ABB RobotStudio station: MinorProjectFINAL.rspag

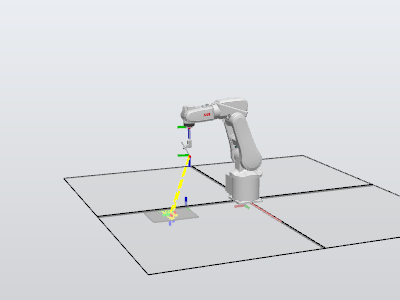
--- station ---
Station Project2 (saved by RobotStudio 23.2.10395.0)
Controller IRB120
  mechanical unit ROB_1: IRB120_3_58__01, 6 joints, base frame (0, 0, 0) mm
Layout (positions relative to the parent item):
  - IRB120_3_58__01 [mechanism, from %ABB.RobotStudio.Models.IRB120%\IRB120_3_58_G_01.rslib] at (0, 0, 0) mm; joint values [-1.5934, 0.3289, -0.2404, 0.0263, 1.472, 1.8577] (rad or m)
  - paperREVISED [part] at (105, -375, -42.57) mm, rotated rx -90 ry 0 rz 180 deg, size 210 x 3 x 297 mm
  - Part_1 [part] at (105, -375, -42.57) mm, rotated rx -90 ry 0 rz 180 deg, size 210 x 0 x 297 mm
  - Penjamin_Franklin [mechanism, from Components\Penjamin_Franklin_And his associates.rslib] at (-7.04, -394.91, 516.59) mm, rotated rx 179.86 ry -1.61 rz -17.87 deg; joint values [-0.07, 0.002] (rad or m)
Attachment: Penjamin_Franklin is attached to IRB120_3_58__01 / Link6

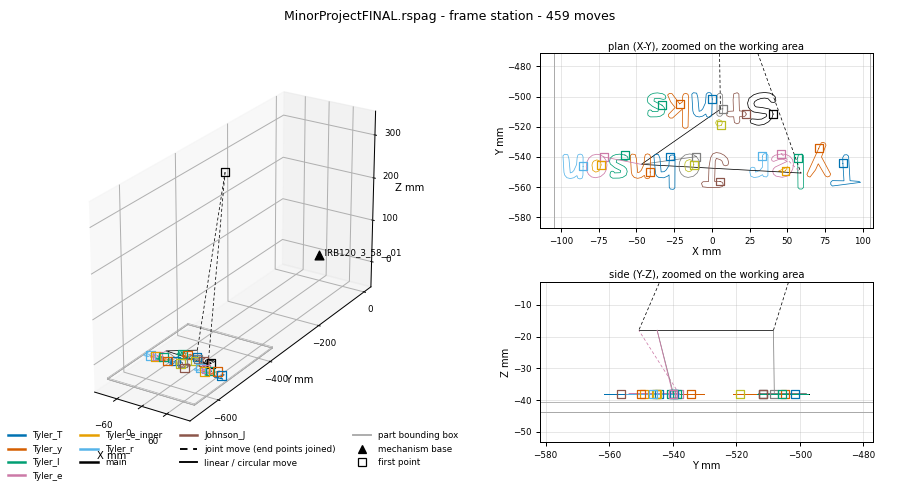
[picture p0: tool path of MinorProjectFINAL.rspag in frame station, 459 of 459 moves have a stored position in this frame; points joined in program order, loops and branches not executed]
--- Controller Data/IRB120/RAPID/TASK1/PROGMOD/CalibData.mod ---
MODULE CalibData
    PERS tooldata TCP_Pen_holder:=[TRUE,[[3.648,-1.274,111.716],[0.96514184,0.252402043,-0.069241872,0.000002181]],[0.3,[0,0,1],[1,0,0,0],0,0,0]];
    TASK PERS wobjdata Workobject_1:=[FALSE,TRUE,"",[[0,-5.508826639,-38],[0.707106781,0,0,-0.707106781]],[[375,-105,-3],[1,0,0,0]]];
    PERS tooldata My_Mechanism_1:=[TRUE,[[6.094876052,-1.40734435,179.947302726],[1,0,0,0]],[1,[1,0,0],[1,0,0,0],0,0,0]];
ENDMODULE

--- Controller Data/IRB120/RAPID/TASK1/PROGMOD/Module1.mod ---
MODULE Module1
    CONST robtarget Target_10:=[[163.751041257,191.907801073,3],[0,0.698319762,0.715785939,0],[0,0,0,0],[9E+09,9E+09,9E+09,9E+09,9E+09,9E+09]];
    CONST robtarget Target_20:=[[175.314304081,192.628796128,3],[0,0.698319762,0.715785939,0],[-1,0,1,0],[9E+09,9E+09,9E+09,9E+09,9E+09,9E+09]];
    CONST robtarget Target_30:=[[175.182166106,184.939790519,3],[0,0.698319762,0.715785939,0],[-1,0,1,0],[9E+09,9E+09,9E+09,9E+09,9E+09,9E+09]];
    CONST robtarget Target_40:=[[176.230100562,183.867034252,3],[0,0.698319762,0.715785939,0],[-1,0,1,0],[9E+09,9E+09,9E+09,9E+09,9E+09,9E+09]];
    CONST robtarget Target_50:=[[177.723746323,183.872070355,3],[0,0.698319762,0.715785939,0],[-1,0,1,0],[9E+09,9E+09,9E+09,9E+09,9E+09,9E+09]];
    CONST robtarget Target_60:=[[178.753770561,184.951832845,3],[0,0.698319762,0.715785939,0],[-1,0,1,0],[9E+09,9E+09,9E+09,9E+09,9E+09,9E+09]];
    CONST robtarget Target_70:=[[179.350705843,202.80856544,3],[0,0.698319762,0.715785939,0],[-1,0,1,0],[9E+09,9E+09,9E+09,9E+09,9E+09,9E+09]];
    CONST robtarget Target_80:=[[178.224639727,203.8775082,3],[0,0.698319762,0.715785939,0],[-1,0,1,0],[9E+09,9E+09,9E+09,9E+09,9E+09,9E+09]];
    CONST robtarget Target_90:=[[176.332276325,203.6047191,3],[0,0.698319762,0.715785939,0],[-1,0,1,0],[9E+09,9E+09,9E+09,9E+09,9E+09,9E+09]];
    CONST robtarget Target_100:=[[175.679129405,202.419661956,3],[0,0.698319762,0.715785939,0],[-1,0,1,0],[9E+09,9E+09,9E+09,9E+09,9E+09,9E+09]];
    CONST robtarget Target_110:=[[175.243917573,196.649555106,3],[0,0.698319762,0.715785939,0],[-1,0,1,0],[9E+09,9E+09,9E+09,9E+09,9E+09,9E+09]];
    CONST robtarget Target_120:=[[158.978457861,195.688923582,3],[0,0.698319762,0.715785939,0],[-1,0,1,0],[9E+09,9E+09,9E+09,9E+09,9E+09,9E+09]];
    CONST robtarget Target_130:=[[157.984185345,194.541790913,3],[0,0.698319762,0.715785939,0],[-1,0,1,0],[9E+09,9E+09,9E+09,9E+09,9E+09,9E+09]];
    CONST robtarget Target_140:=[[158.139068583,192.85150333,3],[0,0.698319762,0.715785939,0],[-1,0,1,0],[9E+09,9E+09,9E+09,9E+09,9E+09,9E+09]];
    CONST robtarget Target_150:=[[159.868914008,191.809461139,3],[0,0.698319762,0.715785939,0],[-1,0,1,0],[9E+09,9E+09,9E+09,9E+09,9E+09,9E+09]];
    CONST robtarget Target_160:=[[163.751041257,191.907801073,3],[0,0.698319762,0.715785939,0],[-1,0,1,0],[9E+09,9E+09,9E+09,9E+09,9E+09,9E+09]];
    CONST robtarget Target_170:=[[153.759568588,175.918000731,3],[0,0.698319762,0.715785939,0],[0,0,0,0],[9E+09,9E+09,9E+09,9E+09,9E+09,9E+09]];
    CONST robtarget Target_180:=[[170.978298864,168.061940799,3],[0,0.698319762,0.715785939,0],[-1,0,1,0],[9E+09,9E+09,9E+09,9E+09,9E+09,9E+09]];
    CONST robtarget Target_190:=[[172.297566022,168.691559399,3],[0,0.698319762,0.715785939,0],[-1,0,1,0],[9E+09,9E+09,9E+09,9E+09,9E+09,9E+09]];
    CONST robtarget Target_200:=[[172.832695065,170.114212978,3],[0,0.698319762,0.715785939,0],[-1,0,1,0],[9E+09,9E+09,9E+09,9E+09,9E+09,9E+09]];
    CONST robtarget Target_210:=[[168.074802834,173.749748589,3],[0,0.698319762,0.715785939,0],[-1,0,1,0],[9E+09,9E+09,9E+09,9E+09,9E+09,9E+09]];
    CONST robtarget Target_220:=[[164.005001441,175.583125337,3],[0,0.698319762,0.715785939,0],[-1,0,1,0],[9E+09,9E+09,9E+09,9E+09,9E+09,9E+09]];
    CONST robtarget Target_230:=[[172.073672363,180.31333522,3],[0,0.698319762,0.715785939,0],[-1,0,1,0],[9E+09,9E+09,9E+09,9E+09,9E+09,9E+09]];
    CONST robtarget Target_240:=[[172.764944958,181.779137598,3],[0,0.698319762,0.715785939,0],[-1,0,1,0],[9E+09,9E+09,9E+09,9E+09,9E+09,9E+09]];
    CONST robtarget Target_250:=[[172.177663158,183.183796934,3],[0,0.698319762,0.715785939,0],[-1,0,1,0],[9E+09,9E+09,9E+09,9E+09,9E+09,9E+09]];
    CONST robtarget Target_260:=[[170.825808862,183.79020191,3],[0,0.698319762,0.715785939,0],[-1,0,1,0],[9E+09,9E+09,9E+09,9E+09,9E+09,9E+09]];
    CONST robtarget Target_270:=[[159.479522834,177.713345848,3],[0,0.698319762,0.715785939,0],[-1,0,1,0],[9E+09,9E+09,9E+09,9E+09,9E+09,9E+09]];
    CONST robtarget Target_280:=[[151.640593909,180.699110514,3],[0,0.698319762,0.715785939,0],[-1,0,1,0],[9E+09,9E+09,9E+09,9E+09,9E+09,9E+09]];
    CONST robtarget Target_290:=[[150.321278848,180.083699197,3],[0,0.698319762,0.715785939,0],[-1,0,1,0],[9E+09,9E+09,9E+09,9E+09,9E+09,9E+09]];
    CONST robtarget Target_300:=[[149.800359463,178.661095912,3],[0,0.698319762,0.715785939,0],[-1,0,1,0],[9E+09,9E+09,9E+09,9E+09,9E+09,9E+09]];
    CONST robtarget Target_310:=[[150.137994684,177.553972625,3],[0,0.698319762,0.715785939,0],[-1,0,1,0],[9E+09,9E+09,9E+09,9E+09,9E+09,9E+09]];
    CONST robtarget Target_320:=[[153.759568588,175.918000731,3],[0,0.698319762,0.715785939,0],[-1,0,1,0],[9E+09,9E+09,9E+09,9E+09,9E+09,9E+09]];
    CONST robtarget Target_330:=[[160.172124107,161.930071278,3],[0,0.698319762,0.715785939,0],[0,0,0,0],[9E+09,9E+09,9E+09,9E+09,9E+09,9E+09]];
    CONST robtarget Target_340:=[[179.798680323,162.131224905,3],[0,0.698319762,0.715785939,0],[-1,0,1,0],[9E+09,9E+09,9E+09,9E+09,9E+09,9E+09]];
    CONST robtarget Target_350:=[[180.757857374,163.153918745,3],[0,0.698319762,0.715785939,0],[-1,0,1,0],[9E+09,9E+09,9E+09,9E+09,9E+09,9E+09]];
    CONST robtarget Target_360:=[[180.758005009,164.688432855,3],[0,0.698319762,0.715785939,0],[-1,0,1,0],[9E+09,9E+09,9E+09,9E+09,9E+09,9E+09]];
    CONST robtarget Target_370:=[[179.791737876,165.768569394,3],[0,0.698319762,0.715785939,0],[-1,0,1,0],[9E+09,9E+09,9E+09,9E+09,9E+09,9E+09]];
    CONST robtarget Target_380:=[[158.617763384,165.707834792,3],[0,0.698319762,0.715785939,0],[-1,0,1,0],[9E+09,9E+09,9E+09,9E+09,9E+09,9E+09]];
    CONST robtarget Target_390:=[[157.598293381,164.660075232,3],[0,0.698319762,0.715785939,0],[-1,0,1,0],[9E+09,9E+09,9E+09,9E+09,9E+09,9E+09]];
    CONST robtarget Target_400:=[[158.145784606,162.413430484,3],[0,0.698319762,0.715785939,0],[-1,0,1,0],[9E+09,9E+09,9E+09,9E+09,9E+09,9E+09]];
    CONST robtarget Target_410:=[[160.172124107,161.930071278,3],[0,0.698319762,0.715785939,0],[-1,0,1,0],[9E+09,9E+09,9E+09,9E+09,9E+09,9E+09]];
    CONST robtarget Target_420:=[[157.466190298,151.165133067,3],[0,0.698319762,0.715785939,0],[0,0,0,0],[9E+09,9E+09,9E+09,9E+09,9E+09,9E+09]];
    CONST robtarget Target_430:=[[158.332912519,146.948141754,3],[0,0.698319762,0.715785939,0],[-1,0,1,0],[9E+09,9E+09,9E+09,9E+09,9E+09,9E+09]];
    CONST robtarget Target_440:=[[159.511105335,145.172500176,3],[0,0.698319762,0.715785939,0],[-1,0,1,0],[9E+09,9E+09,9E+09,9E+09,9E+09,9E+09]];
    CONST robtarget Target_450:=[[160.983662843,144.584262074,3],[0,0.698319762,0.715785939,0],[-1,0,1,0],[9E+09,9E+09,9E+09,9E+09,9E+09,9E+09]];
    CONST robtarget Target_460:=[[162.058689867,144.95730411,3],[0,0.698319762,0.715785939,0],[-1,0,1,0],[9E+09,9E+09,9E+09,9E+09,9E+09,9E+09]];
    CONST robtarget Target_470:=[[162.413713886,146.066767593,3],[0,0.698319762,0.715785939,0],[-1,0,1,0],[9E+09,9E+09,9E+09,9E+09,9E+09,9E+09]];
    CONST robtarget Target_480:=[[161.120102459,149.419153576,3],[0,0.698319762,0.715785939,0],[-1,0,1,0],[9E+09,9E+09,9E+09,9E+09,9E+09,9E+09]];
    CONST robtarget Target_490:=[[161.007182593,152.356373467,3],[0,0.698319762,0.715785939,0],[-1,0,1,0],[9E+09,9E+09,9E+09,9E+09,9E+09,9E+09]];
    CONST robtarget Target_500:=[[162.383437332,155.046418547,3],[0,0.698319762,0.715785939,0],[-1,0,1,0],[9E+09,9E+09,9E+09,9E+09,9E+09,9E+09]];
    CONST robtarget Target_510:=[[166.147149915,147.073948161,3],[0,0.698319762,0.715785939,0],[-1,0,1,0],[9E+09,9E+09,9E+09,9E+09,9E+09,9E+09]];
    CONST robtarget Target_520:=[[167.44807257,145.7676018,3],[0,0.698319762,0.715785939,0],[-1,0,1,0],[9E+09,9E+09,9E+09,9E+09,9E+09,9E+09]];
    CONST robtarget Target_530:=[[168.923660296,145.335667719,3],[0,0.698319762,0.715785939,0],[-1,0,1,0],[9E+09,9E+09,9E+09,9E+09,9E+09,9E+09]];
    CONST robtarget Target_540:=[[170.84708047,145.878521444,3],[0,0.698319762,0.715785939,0],[-1,0,1,0],[9E+09,9E+09,9E+09,9E+09,9E+09,9E+09]];
    CONST robtarget Target_550:=[[172.184335093,147.492140687,3],[0,0.698319762,0.715785939,0],[-1,0,1,0],[9E+09,9E+09,9E+09,9E+09,9E+09,9E+09]];
    CONST robtarget Target_560:=[[172.966155304,151.601026046,3],[0,0.698319762,0.715785939,0],[-1,0,1,0],[9E+09,9E+09,9E+09,9E+09,9E+09,9E+09]];
    CONST robtarget Target_570:=[[172.266262418,154.799124826,3],[0,0.698319762,0.715785939,0],[-1,0,1,0],[9E+09,9E+09,9E+09,9E+09,9E+09,9E+09]];
    CONST robtarget Target_580:=[[170.190632557,157.260845666,3],[0,0.698319762,0.715785939,0],[-1,0,1,0],[9E+09,9E+09,9E+09,9E+09,9E+09,9E+09]];
    CONST robtarget Target_590:=[[167.422340833,158.668803926,3],[0,0.698319762,0.715785939,0],[-1,0,1,0],[9E+09,9E+09,9E+09,9E+09,9E+09,9E+09]];
    CONST robtarget Target_600:=[[164.103105526,159.130046378,3],[0,0.698319762,0.715785939,0],[-1,0,1,0],[9E+09,9E+09,9E+09,9E+09,9E+09,9E+09]];
    CONST robtarget Target_610:=[[161.217274645,158.523560707,3],[0,0.698319762,0.715785939,0],[-1,0,1,0],[9E+09,9E+09,9E+09,9E+09,9E+09,9E+09]];
    CONST robtarget Target_620:=[[159.067198932,156.726044653,3],[0,0.698319762,0.715785939,0],[-1,0,1,0],[9E+09,9E+09,9E+09,9E+09,9E+09,9E+09]];
    CONST robtarget Target_630:=[[157.860720068,154.253257576,3],[0,0.698319762,0.715785939,0],[-1,0,1,0],[9E+09,9E+09,9E+09,9E+09,9E+09,9E+09]];
    CONST robtarget Target_640:=[[157.466190298,151.165133067,3],[0,0.698319762,0.715785939,0],[-1,0,1,0],[9E+09,9E+09,9E+09,9E+09,9E+09,9E+09]];
    CONST robtarget Target_650:=[[168.639209719,153.845580268,3],[0,0.698319762,0.715785939,0],[0,0,0,0],[9E+09,9E+09,9E+09,9E+09,9E+09,9E+09]];
    CONST robtarget Target_660:=[[169.527749784,151.589432826,3],[0,0.698319762,0.715785939,0],[-1,0,1,0],[9E+09,9E+09,9E+09,9E+09,9E+09,9E+09]];
    CONST robtarget Target_670:=[[168.996213692,149.10115439,3],[0,0.698319762,0.715785939,0],[-1,0,1,0],[9E+09,9E+09,9E+09,9E+09,9E+09,9E+09]];
    CONST robtarget Target_680:=[[165.991391199,155.342751383,3],[0,0.698319762,0.715785939,0],[-1,0,1,0],[9E+09,9E+09,9E+09,9E+09,9E+09,9E+09]];
    CONST robtarget Target_690:=[[168.639209719,153.845580268,3],[0,0.698319762,0.715785939,0],[-1,0,1,0],[9E+09,9E+09,9E+09,9E+09,9E+09,9E+09]];
    CONST robtarget Target_700:=[[159.08585114,138.553482656,3],[0,0.698319762,0.715785939,0],[0,0,0,0],[9E+09,9E+09,9E+09,9E+09,9E+09,9E+09]];
    CONST robtarget Target_710:=[[166.232578876,138.591784231,3],[0,0.698319762,0.715785939,0],[-1,0,1,0],[9E+09,9E+09,9E+09,9E+09,9E+09,9E+09]];
    CONST robtarget Target_720:=[[168.444594894,136.76635106,3],[0,0.698319762,0.715785939,0],[-1,0,1,0],[9E+09,9E+09,9E+09,9E+09,9E+09,9E+09]];
    CONST robtarget Target_730:=[[169.530122845,134.02777656,3],[0,0.698319762,0.715785939,0],[-1,0,1,0],[9E+09,9E+09,9E+09,9E+09,9E+09,9E+09]];
    CONST robtarget Target_740:=[[166.711519604,133.499671613,3],[0,0.698319762,0.715785939,0],[-1,0,1,0],[9E+09,9E+09,9E+09,9E+09,9E+09,9E+09]];
    CONST robtarget Target_750:=[[166.254280251,132.15542517,3],[0,0.698319762,0.715785939,0],[-1,0,1,0],[9E+09,9E+09,9E+09,9E+09,9E+09,9E+09]];
    CONST robtarget Target_760:=[[166.802526185,130.739972078,3],[0,0.698319762,0.715785939,0],[-1,0,1,0],[9E+09,9E+09,9E+09,9E+09,9E+09,9E+09]];
    CONST robtarget Target_770:=[[169.386818084,130.176801905,3],[0,0.698319762,0.715785939,0],[-1,0,1,0],[9E+09,9E+09,9E+09,9E+09,9E+09,9E+09]];
    CONST robtarget Target_780:=[[172.218984231,130.896775724,3],[0,0.698319762,0.715785939,0],[-1,0,1,0],[9E+09,9E+09,9E+09,9E+09,9E+09,9E+09]];
    CONST robtarget Target_790:=[[173.156645819,133.031201627,3],[0,0.698319762,0.715785939,0],[-1,0,1,0],[9E+09,9E+09,9E+09,9E+09,9E+09,9E+09]];
    CONST robtarget Target_800:=[[172.677884374,135.960083101,3],[0,0.698319762,0.715785939,0],[-1,0,1,0],[9E+09,9E+09,9E+09,9E+09,9E+09,9E+09]];
    CONST robtarget Target_810:=[[171.262323998,138.608742947,3],[0,0.698319762,0.715785939,0],[-1,0,1,0],[9E+09,9E+09,9E+09,9E+09,9E+09,9E+09]];
    CONST robtarget Target_820:=[[172.475042596,139.230902153,3],[0,0.698319762,0.715785939,0],[-1,0,1,0],[9E+09,9E+09,9E+09,9E+09,9E+09,9E+09]];
    CONST robtarget Target_830:=[[172.739912492,141.268936192,3],[0,0.698319762,0.715785939,0],[-1,0,1,0],[9E+09,9E+09,9E+09,9E+09,9E+09,9E+09]];
    CONST robtarget Target_840:=[[171.738633757,142.199761024,3],[0,0.698319762,0.715785939,0],[-1,0,1,0],[9E+09,9E+09,9E+09,9E+09,9E+09,9E+09]];
    CONST robtarget Target_850:=[[158.348865178,142.216780556,3],[0,0.698319762,0.715785939,0],[-1,0,1,0],[9E+09,9E+09,9E+09,9E+09,9E+09,9E+09]];
    CONST robtarget Target_860:=[[157.343188099,141.289841504,3],[0,0.698319762,0.715785939,0],[-1,0,1,0],[9E+09,9E+09,9E+09,9E+09,9E+09,9E+09]];
    CONST robtarget Target_870:=[[157.339567123,139.730448483,3],[0,0.698319762,0.715785939,0],[-1,0,1,0],[9E+09,9E+09,9E+09,9E+09,9E+09,9E+09]];
    CONST robtarget Target_880:=[[158.344774317,138.689520265,3],[0,0.698319762,0.715785939,0],[-1,0,1,0],[9E+09,9E+09,9E+09,9E+09,9E+09,9E+09]];
    CONST robtarget Target_890:=[[159.08585114,138.553482656,3],[0,0.698319762,0.715785939,0],[-1,0,1,0],[9E+09,9E+09,9E+09,9E+09,9E+09,9E+09]];
    CONST robtarget Homes:=[[3.863516215,-397.404717523,336.886300892],[0.003386746,0.987758585,-0.155352434,0.013679542],[-2,0,1,0],[9E+09,9E+09,9E+09,9E+09,9E+09,9E+09]];
    CONST robtarget liftPoint_Tyler:=[[170.167,164.128,23],[0,0.698319762,0.715785939,0],[-1,0,1,0],[9E+09,9E+09,9E+09,9E+09,9E+09,9E+09]];
    CONST robtarget Target_900:=[[175.775906994,110.505400925,3],[0,0.698319762,0.715785939,0],[-2,1,-1,0],[9E+09,9E+09,9E+09,9E+09,9E+09,9E+09]];
    CONST robtarget Target_910:=[[175.731485499,106.825258538,3],[0,0.698319762,0.715785939,0],[-2,1,-1,0],[9E+09,9E+09,9E+09,9E+09,9E+09,9E+09]];
    CONST robtarget Target_920:=[[162.3172094,107.263116295,3],[0,0.698319762,0.715785939,0],[-2,1,-1,0],[9E+09,9E+09,9E+09,9E+09,9E+09,9E+09]];
    CONST robtarget Target_930:=[[160.425013825,107.99558071,3],[0,0.698319762,0.715785939,0],[-2,1,-1,0],[9E+09,9E+09,9E+09,9E+09,9E+09,9E+09]];
    CONST robtarget Target_940:=[[161.374954401,110.705498367,3],[0,0.698319762,0.715785939,0],[-2,1,-1,0],[9E+09,9E+09,9E+09,9E+09,9E+09,9E+09]];
    CONST robtarget Target_950:=[[162.300171542,111.790233782,3],[0,0.698319762,0.715785939,0],[-2,1,-1,0],[9E+09,9E+09,9E+09,9E+09,9E+09,9E+09]];
    CONST robtarget Target_960:=[[164.806818321,112.660077554,3],[0,0.698319762,0.715785939,0],[-2,1,-1,0],[9E+09,9E+09,9E+09,9E+09,9E+09,9E+09]];
    CONST robtarget Target_970:=[[165.348767223,114.164446335,3],[0,0.698319762,0.715785939,0],[-2,1,-1,0],[9E+09,9E+09,9E+09,9E+09,9E+09,9E+09]];
    CONST robtarget Target_980:=[[164.789571873,115.665102404,3],[0,0.698319762,0.715785939,0],[-2,1,-1,0],[9E+09,9E+09,9E+09,9E+09,9E+09,9E+09]];
    CONST robtarget Target_990:=[[163.125514309,116.16034525,3],[0,0.698319762,0.715785939,0],[-2,1,-1,0],[9E+09,9E+09,9E+09,9E+09,9E+09,9E+09]];
    CONST robtarget Target_1000:=[[160.563384619,115.419967167,3],[0,0.698319762,0.715785939,0],[-2,1,-1,0],[9E+09,9E+09,9E+09,9E+09,9E+09,9E+09]];
    CONST robtarget Target_1010:=[[158.361392746,113.217334114,3],[0,0.698319762,0.715785939,0],[-2,1,-1,0],[9E+09,9E+09,9E+09,9E+09,9E+09,9E+09]];
    CONST robtarget Target_1020:=[[157.00616506,110.612614131,3],[0,0.698319762,0.715785939,0],[-2,1,-1,0],[9E+09,9E+09,9E+09,9E+09,9E+09,9E+09]];
    CONST robtarget Target_1030:=[[156.560356456,107.982550303,3],[0,0.698319762,0.715785939,0],[-2,1,-1,0],[9E+09,9E+09,9E+09,9E+09,9E+09,9E+09]];
    CONST robtarget Target_1040:=[[157.424300306,105.644618187,3],[0,0.698319762,0.715785939,0],[-2,1,-1,0],[9E+09,9E+09,9E+09,9E+09,9E+09,9E+09]];
    CONST robtarget Target_1050:=[[159.997448553,104.172057738,3],[0,0.698319762,0.715785939,0],[-2,1,-1,0],[9E+09,9E+09,9E+09,9E+09,9E+09,9E+09]];
    CONST robtarget Target_1060:=[[166.0289515,103.116099725,3],[0,0.698319762,0.715785939,0],[-2,1,-1,0],[9E+09,9E+09,9E+09,9E+09,9E+09,9E+09]];
    CONST robtarget Target_1070:=[[175.830387142,102.776182007,3],[0,0.698319762,0.715785939,0],[-2,1,-1,0],[9E+09,9E+09,9E+09,9E+09,9E+09,9E+09]];
    CONST robtarget Target_1080:=[[175.902977488,99.156821148,3],[0,0.698319762,0.715785939,0],[-2,1,-1,0],[9E+09,9E+09,9E+09,9E+09,9E+09,9E+09]];
    CONST robtarget Target_1090:=[[177.007630849,98.11977592,3],[0,0.698319762,0.715785939,0],[-2,1,-1,0],[9E+09,9E+09,9E+09,9E+09,9E+09,9E+09]];
    CONST robtarget Target_1100:=[[179.292389298,98.951563604,3],[0,0.698319762,0.715785939,0],[-2,1,-1,0],[9E+09,9E+09,9E+09,9E+09,9E+09,9E+09]];
    CONST robtarget Target_1110:=[[179.783379524,102.926267927,3],[0,0.698319762,0.715785939,0],[-2,1,-1,0],[9E+09,9E+09,9E+09,9E+09,9E+09,9E+09]];
    CONST robtarget Target_1120:=[[179.656450737,110.021188597,3],[0,0.698319762,0.715785939,0],[-2,1,-1,0],[9E+09,9E+09,9E+09,9E+09,9E+09,9E+09]];
    CONST robtarget Target_1130:=[[179.166938366,111.927031105,3],[0,0.698319762,0.715785939,0],[-2,1,-1,0],[9E+09,9E+09,9E+09,9E+09,9E+09,9E+09]];
    CONST robtarget Target_1140:=[[177.715551642,112.557965304,3],[0,0.698319762,0.715785939,0],[-2,1,-1,0],[9E+09,9E+09,9E+09,9E+09,9E+09,9E+09]];
    CONST robtarget Target_1150:=[[176.282616704,111.927958684,3],[0,0.698319762,0.715785939,0],[-2,1,-1,0],[9E+09,9E+09,9E+09,9E+09,9E+09,9E+09]];
    CONST robtarget Target_1160:=[[175.775906994,110.505400925,3],[0,0.698319762,0.715785939,0],[-2,1,-1,0],[9E+09,9E+09,9E+09,9E+09,9E+09,9E+09]];
    CONST robtarget Target_1170:=[[159.276068814,94.777825568,3],[0,0.698319762,0.715785939,0],[-2,1,-1,0],[9E+09,9E+09,9E+09,9E+09,9E+09,9E+09]];
    CONST robtarget Target_1180:=[[157.929711577,92.698841911,3],[0,0.698319762,0.715785939,0],[-2,1,-1,0],[9E+09,9E+09,9E+09,9E+09,9E+09,9E+09]];
    CONST robtarget Target_1190:=[[157.486846922,90.253496701,3],[0,0.698319762,0.715785939,0],[-2,1,-1,0],[9E+09,9E+09,9E+09,9E+09,9E+09,9E+09]];
    CONST robtarget Target_1200:=[[158.146958921,87.268396908,3],[0,0.698319762,0.715785939,0],[-2,1,-1,0],[9E+09,9E+09,9E+09,9E+09,9E+09,9E+09]];
    CONST robtarget Target_1210:=[[160.104836866,84.962563313,3],[0,0.698319762,0.715785939,0],[-2,1,-1,0],[9E+09,9E+09,9E+09,9E+09,9E+09,9E+09]];
    CONST robtarget Target_1220:=[[162.680993817,83.649859269,3],[0,0.698319762,0.715785939,0],[-2,1,-1,0],[9E+09,9E+09,9E+09,9E+09,9E+09,9E+09]];
    CONST robtarget Target_1230:=[[165.737271089,83.219707087,3],[0,0.698319762,0.715785939,0],[-2,1,-1,0],[9E+09,9E+09,9E+09,9E+09,9E+09,9E+09]];
    CONST robtarget Target_1240:=[[168.517281523,83.60561224,3],[0,0.698319762,0.715785939,0],[-2,1,-1,0],[9E+09,9E+09,9E+09,9E+09,9E+09,9E+09]];
    CONST robtarget Target_1250:=[[170.804557641,84.742891106,3],[0,0.698319762,0.715785939,0],[-2,1,-1,0],[9E+09,9E+09,9E+09,9E+09,9E+09,9E+09]];
    CONST robtarget Target_1260:=[[172.502920539,86.716487904,3],[0,0.698319762,0.715785939,0],[-2,1,-1,0],[9E+09,9E+09,9E+09,9E+09,9E+09,9E+09]];
    CONST robtarget Target_1270:=[[173.062650846,89.26880086,3],[0,0.698319762,0.715785939,0],[-2,1,-1,0],[9E+09,9E+09,9E+09,9E+09,9E+09,9E+09]];
    CONST robtarget Target_1280:=[[172.326476842,92.694110719,3],[0,0.698319762,0.715785939,0],[-2,1,-1,0],[9E+09,9E+09,9E+09,9E+09,9E+09,9E+09]];
    CONST robtarget Target_1290:=[[170.143891247,95.269135257,3],[0,0.698319762,0.715785939,0],[-2,1,-1,0],[9E+09,9E+09,9E+09,9E+09,9E+09,9E+09]];
    CONST robtarget Target_1300:=[[167.510845294,96.599405006,3],[0,0.698319762,0.715785939,0],[-2,1,-1,0],[9E+09,9E+09,9E+09,9E+09,9E+09,9E+09]];
    CONST robtarget Target_1310:=[[164.540029593,96.969467873,3],[0,0.698319762,0.715785939,0],[-2,1,-1,0],[9E+09,9E+09,9E+09,9E+09,9E+09,9E+09]];
    CONST robtarget Target_1320:=[[161.576033584,96.366266342,3],[0,0.698319762,0.715785939,0],[-2,1,-1,0],[9E+09,9E+09,9E+09,9E+09,9E+09,9E+09]];
    CONST robtarget Target_1330:=[[159.276068814,94.777825568,3],[0,0.698319762,0.715785939,0],[-2,1,-1,0],[9E+09,9E+09,9E+09,9E+09,9E+09,9E+09]];
    CONST robtarget Target_1340:=[[164.553299553,93.033762171,3],[0,0.698319762,0.715785939,0],[-2,1,-1,0],[9E+09,9E+09,9E+09,9E+09,9E+09,9E+09]];
    CONST robtarget Target_1350:=[[167.710414693,92.191903115,3],[0,0.698319762,0.715785939,0],[-2,1,-1,0],[9E+09,9E+09,9E+09,9E+09,9E+09,9E+09]];
    CONST robtarget Target_1360:=[[168.915041174,91.002453619,3],[0,0.698319762,0.715785939,0],[-2,1,-1,0],[9E+09,9E+09,9E+09,9E+09,9E+09,9E+09]];
    CONST robtarget Target_1370:=[[169.3110385,89.440860296,3],[0,0.698319762,0.715785939,0],[-2,1,-1,0],[9E+09,9E+09,9E+09,9E+09,9E+09,9E+09]];
    CONST robtarget Target_1380:=[[168.162996215,87.543715835,3],[0,0.698319762,0.715785939,0],[-2,1,-1,0],[9E+09,9E+09,9E+09,9E+09,9E+09,9E+09]];
    CONST robtarget Target_1390:=[[164.729851,87.024181912,3],[0,0.698319762,0.715785939,0],[-2,1,-1,0],[9E+09,9E+09,9E+09,9E+09,9E+09,9E+09]];
    CONST robtarget Target_1400:=[[163.226272679,87.33169039,3],[0,0.698319762,0.715785939,0],[-2,1,-1,0],[9E+09,9E+09,9E+09,9E+09,9E+09,9E+09]];
    CONST robtarget Target_1410:=[[162.06916418,88.1234726,3],[0,0.698319762,0.715785939,0],[-2,1,-1,0],[9E+09,9E+09,9E+09,9E+09,9E+09,9E+09]];
    CONST robtarget Target_1420:=[[161.223636366,90.266095978,3],[0,0.698319762,0.715785939,0],[-2,1,-1,0],[9E+09,9E+09,9E+09,9E+09,9E+09,9E+09]];
    CONST robtarget Target_1430:=[[161.942226456,92.058785513,3],[0,0.698319762,0.715785939,0],[-2,1,-1,0],[9E+09,9E+09,9E+09,9E+09,9E+09,9E+09]];
    CONST robtarget Target_1440:=[[163.0480419,92.787138913,3],[0,0.698319762,0.715785939,0],[-2,1,-1,0],[9E+09,9E+09,9E+09,9E+09,9E+09,9E+09]];
    CONST robtarget Target_1450:=[[164.553299553,93.033762171,3],[0,0.698319762,0.715785939,0],[-2,1,-1,0],[9E+09,9E+09,9E+09,9E+09,9E+09,9E+09]];
    CONST robtarget Target_1460:=[[159.19401738,76.974331877,3],[0,0.698319762,0.715785939,0],[-2,1,-1,0],[9E+09,9E+09,9E+09,9E+09,9E+09,9E+09]];
    CONST robtarget Target_1470:=[[165.390517427,76.497928224,3],[0,0.698319762,0.715785939,0],[-2,1,-1,0],[9E+09,9E+09,9E+09,9E+09,9E+09,9E+09]];
    CONST robtarget Target_1480:=[[168.152961856,74.716975641,3],[0,0.698319762,0.715785939,0],[-2,1,-1,0],[9E+09,9E+09,9E+09,9E+09,9E+09,9E+09]];
    CONST robtarget Target_1490:=[[169.244459454,73.367307985,3],[0,0.698319762,0.715785939,0],[-2,1,-1,0],[9E+09,9E+09,9E+09,9E+09,9E+09,9E+09]];
    CONST robtarget Target_1500:=[[169.418127554,71.375151118,3],[0,0.698319762,0.715785939,0],[-2,1,-1,0],[9E+09,9E+09,9E+09,9E+09,9E+09,9E+09]];
    CONST robtarget Target_1510:=[[160.31671931,70.584304991,3],[0,0.698319762,0.715785939,0],[-2,1,-1,0],[9E+09,9E+09,9E+09,9E+09,9E+09,9E+09]];
    CONST robtarget Target_1520:=[[157.86917958,69.570807458,3],[0,0.698319762,0.715785939,0],[-2,1,-1,0],[9E+09,9E+09,9E+09,9E+09,9E+09,9E+09]];
    CONST robtarget Target_1530:=[[157.650162968,67.628834824,3],[0,0.698319762,0.715785939,0],[-2,1,-1,0],[9E+09,9E+09,9E+09,9E+09,9E+09,9E+09]];
    CONST robtarget Target_1540:=[[158.630714107,66.523869711,3],[0,0.698319762,0.715785939,0],[-2,1,-1,0],[9E+09,9E+09,9E+09,9E+09,9E+09,9E+09]];
    CONST robtarget Target_1550:=[[170.77309542,67.735242064,3],[0,0.698319762,0.715785939,0],[-2,1,-1,0],[9E+09,9E+09,9E+09,9E+09,9E+09,9E+09]];
    CONST robtarget Target_1560:=[[172.067452503,68.378991271,3],[0,0.698319762,0.715785939,0],[-2,1,-1,0],[9E+09,9E+09,9E+09,9E+09,9E+09,9E+09]];
    CONST robtarget Target_1570:=[[173.085710436,69.789063982,3],[0,0.698319762,0.715785939,0],[-2,1,-1,0],[9E+09,9E+09,9E+09,9E+09,9E+09,9E+09]];
    CONST robtarget Target_1580:=[[173.289145178,73.187338868,3],[0,0.698319762,0.715785939,0],[-2,1,-1,0],[9E+09,9E+09,9E+09,9E+09,9E+09,9E+09]];
    CONST robtarget Target_1590:=[[172.26880383,75.560268231,3],[0,0.698319762,0.715785939,0],[-2,1,-1,0],[9E+09,9E+09,9E+09,9E+09,9E+09,9E+09]];
    CONST robtarget Target_1600:=[[171.371831589,76.63176442,3],[0,0.698319762,0.715785939,0],[-2,1,-1,0],[9E+09,9E+09,9E+09,9E+09,9E+09,9E+09]];
    CONST robtarget Target_1610:=[[179.626520965,76.759055892,3],[0,0.698319762,0.715785939,0],[-2,0,-1,0],[9E+09,9E+09,9E+09,9E+09,9E+09,9E+09]];
    CONST robtarget Target_1620:=[[180.753677289,77.476828643,3],[0,0.698319762,0.715785939,0],[-2,0,-1,0],[9E+09,9E+09,9E+09,9E+09,9E+09,9E+09]];
    CONST robtarget Target_1630:=[[180.994004844,79.417099286,3],[0,0.698319762,0.715785939,0],[-2,0,-1,0],[9E+09,9E+09,9E+09,9E+09,9E+09,9E+09]];
    CONST robtarget Target_1640:=[[180.009982837,80.493623504,3],[0,0.698319762,0.715785939,0],[-2,0,-1,0],[9E+09,9E+09,9E+09,9E+09,9E+09,9E+09]];
    CONST robtarget Target_1650:=[[159.144449473,80.613311259,3],[0,0.698319762,0.715785939,0],[-2,1,-1,0],[9E+09,9E+09,9E+09,9E+09,9E+09,9E+09]];
    CONST robtarget Target_1660:=[[158.153655217,79.483941873,3],[0,0.698319762,0.715785939,0],[-2,1,-1,0],[9E+09,9E+09,9E+09,9E+09,9E+09,9E+09]];
    CONST robtarget Target_1670:=[[158.317789462,77.688907073,3],[0,0.698319762,0.715785939,0],[-2,1,-1,0],[9E+09,9E+09,9E+09,9E+09,9E+09,9E+09]];
    CONST robtarget Target_1680:=[[159.19401738,76.974331877,3],[0,0.698319762,0.715785939,0],[-2,1,-1,0],[9E+09,9E+09,9E+09,9E+09,9E+09,9E+09]];
    CONST robtarget Target_1690:=[[169.48675747,64.121961466,3],[0,0.698319762,0.715785939,0],[-2,1,-1,0],[9E+09,9E+09,9E+09,9E+09,9E+09,9E+09]];
    CONST robtarget Target_1700:=[[159.313738911,64.314999427,3],[0,0.698319762,0.715785939,0],[-2,0,0,0],[9E+09,9E+09,9E+09,9E+09,9E+09,9E+09]];
    CONST robtarget Target_1710:=[[157.948274945,63.756259901,3],[0,0.698319762,0.715785939,0],[-2,0,0,0],[9E+09,9E+09,9E+09,9E+09,9E+09,9E+09]];
    CONST robtarget Target_1720:=[[157.410437254,62.347807017,3],[0,0.698319762,0.715785939,0],[-2,0,0,0],[9E+09,9E+09,9E+09,9E+09,9E+09,9E+09]];
    CONST robtarget Target_1730:=[[157.961112555,60.935928878,3],[0,0.698319762,0.715785939,0],[-2,0,0,0],[9E+09,9E+09,9E+09,9E+09,9E+09,9E+09]];
    CONST robtarget Target_1740:=[[159.849926153,60.357968251,3],[0,0.698319762,0.715785939,0],[-2,0,0,0],[9E+09,9E+09,9E+09,9E+09,9E+09,9E+09]];
    CONST robtarget Target_1750:=[[164.36181293,60.013090517,3],[0,0.698319762,0.715785939,0],[-2,0,0,0],[9E+09,9E+09,9E+09,9E+09,9E+09,9E+09]];
    CONST robtarget Target_1760:=[[168.334661535,58.194362031,3],[0,0.698319762,0.715785939,0],[-2,0,0,0],[9E+09,9E+09,9E+09,9E+09,9E+09,9E+09]];
    CONST robtarget Target_1770:=[[169.512242363,57.016017545,3],[0,0.698319762,0.715785939,0],[-2,0,0,0],[9E+09,9E+09,9E+09,9E+09,9E+09,9E+09]];
    CONST robtarget Target_1780:=[[169.907511332,55.81187047,3],[0,0.698319762,0.715785939,0],[-2,0,0,0],[9E+09,9E+09,9E+09,9E+09,9E+09,9E+09]];
    CONST robtarget Target_1790:=[[160.621604004,54.956028888,3],[0,0.698319762,0.715785939,0],[-2,0,0,0],[9E+09,9E+09,9E+09,9E+09,9E+09,9E+09]];
    CONST robtarget Target_1800:=[[157.867842537,54.161722596,3],[0,0.698319762,0.715785939,0],[-2,0,0,0],[9E+09,9E+09,9E+09,9E+09,9E+09,9E+09]];
    CONST robtarget Target_1810:=[[157.57665402,52.029476397,3],[0,0.698319762,0.715785939,0],[-2,0,0,0],[9E+09,9E+09,9E+09,9E+09,9E+09,9E+09]];
    CONST robtarget Target_1820:=[[158.56772102,50.970723913,3],[0,0.698319762,0.715785939,0],[-2,0,0,0],[9E+09,9E+09,9E+09,9E+09,9E+09,9E+09]];
    CONST robtarget Target_1830:=[[169.548626817,51.632923283,3],[0,0.698319762,0.715785939,0],[-2,0,0,0],[9E+09,9E+09,9E+09,9E+09,9E+09,9E+09]];
    CONST robtarget Target_1840:=[[171.425954171,52.150759167,3],[0,0.698319762,0.715785939,0],[-2,0,0,0],[9E+09,9E+09,9E+09,9E+09,9E+09,9E+09]];
    CONST robtarget Target_1850:=[[173.104796596,53.595026505,3],[0,0.698319762,0.715785939,0],[-2,0,0,0],[9E+09,9E+09,9E+09,9E+09,9E+09,9E+09]];
    CONST robtarget Target_1860:=[[173.658368222,55.866698432,3],[0,0.698319762,0.715785939,0],[-2,0,0,0],[9E+09,9E+09,9E+09,9E+09,9E+09,9E+09]];
    CONST robtarget Target_1870:=[[173.128646274,58.109855405,3],[0,0.698319762,0.715785939,0],[-2,0,0,0],[9E+09,9E+09,9E+09,9E+09,9E+09,9E+09]];
    CONST robtarget Target_1880:=[[171.711231833,60.250550561,3],[0,0.698319762,0.715785939,0],[-2,0,0,0],[9E+09,9E+09,9E+09,9E+09,9E+09,9E+09]];
    CONST robtarget Target_1890:=[[173.382360872,60.817425607,3],[0,0.698319762,0.715785939,0],[-2,0,0,0],[9E+09,9E+09,9E+09,9E+09,9E+09,9E+09]];
    CONST robtarget Target_1900:=[[173.935223307,62.247234355,3],[0,0.698319762,0.715785939,0],[-2,0,0,0],[9E+09,9E+09,9E+09,9E+09,9E+09,9E+09]];
    CONST robtarget Target_1910:=[[173.402314827,63.659181935,3],[0,0.698319762,0.715785939,0],[-2,0,0,0],[9E+09,9E+09,9E+09,9E+09,9E+09,9E+09]];
    CONST robtarget Target_1920:=[[171.53202662,64.215880745,3],[0,0.698319762,0.715785939,0],[-2,0,0,0],[9E+09,9E+09,9E+09,9E+09,9E+09,9E+09]];
    CONST robtarget Target_1930:=[[169.48675747,64.121961466,3],[0,0.698319762,0.715785939,0],[-2,0,0,0],[9E+09,9E+09,9E+09,9E+09,9E+09,9E+09]];
    CONST robtarget Target_1940:=[[158.199861844,47.346320771,3],[0,0.698319762,0.715785939,0],[-2,1,-1,0],[9E+09,9E+09,9E+09,9E+09,9E+09,9E+09]];
    CONST robtarget Target_1950:=[[157.628963899,43.891731909,3],[0,0.698319762,0.715785939,0],[-2,1,-1,0],[9E+09,9E+09,9E+09,9E+09,9E+09,9E+09]];
    CONST robtarget Target_1960:=[[157.889451747,41.431010202,3],[0,0.698319762,0.715785939,0],[-2,1,-1,0],[9E+09,9E+09,9E+09,9E+09,9E+09,9E+09]];
    CONST robtarget Target_1970:=[[158.652931475,39.391107595,3],[0,0.698319762,0.715785939,0],[-2,1,-1,0],[9E+09,9E+09,9E+09,9E+09,9E+09,9E+09]];
    CONST robtarget Target_1980:=[[160.218043244,37.691376952,3],[0,0.698319762,0.715785939,0],[-2,1,-1,0],[9E+09,9E+09,9E+09,9E+09,9E+09,9E+09]];
    CONST robtarget Target_1990:=[[162.368966498,37.130293285,3],[0,0.698319762,0.715785939,0],[-2,1,-1,0],[9E+09,9E+09,9E+09,9E+09,9E+09,9E+09]];
    CONST robtarget Target_2000:=[[164.146814192,37.65135098,3],[0,0.698319762,0.715785939,0],[-2,0,-1,0],[9E+09,9E+09,9E+09,9E+09,9E+09,9E+09]];
    CONST robtarget Target_2010:=[[166.591204245,40.654032626,3],[0,0.698319762,0.715785939,0],[-2,0,-1,0],[9E+09,9E+09,9E+09,9E+09,9E+09,9E+09]];
    CONST robtarget Target_2020:=[[168.570761932,44.56446156,3],[0,0.698319762,0.715785939,0],[-2,0,-1,0],[9E+09,9E+09,9E+09,9E+09,9E+09,9E+09]];
    CONST robtarget Target_2030:=[[169.925253649,44.228030753,3],[0,0.698319762,0.715785939,0],[-2,0,-1,0],[9E+09,9E+09,9E+09,9E+09,9E+09,9E+09]];
    CONST robtarget Target_2040:=[[170.072823228,40.495253612,3],[0,0.698319762,0.715785939,0],[-2,0,-1,0],[9E+09,9E+09,9E+09,9E+09,9E+09,9E+09]];
    CONST robtarget Target_2050:=[[169.190256749,39.927508735,3],[0,0.698319762,0.715785939,0],[-2,0,-1,0],[9E+09,9E+09,9E+09,9E+09,9E+09,9E+09]];
    CONST robtarget Target_2060:=[[168.899236118,38.800498766,3],[0,0.698319762,0.715785939,0],[-2,0,-1,0],[9E+09,9E+09,9E+09,9E+09,9E+09,9E+09]];
    CONST robtarget Target_2070:=[[169.54208954,37.768991872,3],[0,0.698319762,0.715785939,0],[-2,0,-1,0],[9E+09,9E+09,9E+09,9E+09,9E+09,9E+09]];
    CONST robtarget Target_2080:=[[171.461375012,37.430917682,3],[0,0.698319762,0.715785939,0],[-2,0,-1,0],[9E+09,9E+09,9E+09,9E+09,9E+09,9E+09]];
    CONST robtarget Target_2090:=[[172.586600524,37.669145141,3],[0,0.698319762,0.715785939,0],[-2,0,-1,0],[9E+09,9E+09,9E+09,9E+09,9E+09,9E+09]];
    CONST robtarget Target_2100:=[[173.565226295,39.242449563,3],[0,0.698319762,0.715785939,0],[-2,0,-1,0],[9E+09,9E+09,9E+09,9E+09,9E+09,9E+09]];
    CONST robtarget Target_2110:=[[173.497108354,43.639751601,3],[0,0.698319762,0.715785939,0],[-2,0,-1,0],[9E+09,9E+09,9E+09,9E+09,9E+09,9E+09]];
    CONST robtarget Target_2120:=[[173.052668328,45.87610074,3],[0,0.698319762,0.715785939,0],[-2,0,-1,0],[9E+09,9E+09,9E+09,9E+09,9E+09,9E+09]];
    CONST robtarget Target_2130:=[[171.585119959,48.14094855,3],[0,0.698319762,0.715785939,0],[-2,0,-1,0],[9E+09,9E+09,9E+09,9E+09,9E+09,9E+09]];
    CONST robtarget Target_2140:=[[169.192007177,48.889472011,3],[0,0.698319762,0.715785939,0],[-2,0,-1,0],[9E+09,9E+09,9E+09,9E+09,9E+09,9E+09]];
    CONST robtarget Target_2150:=[[167.328853508,48.382355593,3],[0,0.698319762,0.715785939,0],[-2,0,-1,0],[9E+09,9E+09,9E+09,9E+09,9E+09,9E+09]];
    CONST robtarget Target_2160:=[[165.774565999,46.874573525,3],[0,0.698319762,0.715785939,0],[-2,1,-1,0],[9E+09,9E+09,9E+09,9E+09,9E+09,9E+09]];
    CONST robtarget Target_2170:=[[163.08914292,41.611926335,3],[0,0.698319762,0.715785939,0],[-2,1,-1,0],[9E+09,9E+09,9E+09,9E+09,9E+09,9E+09]];
    CONST robtarget Target_2180:=[[161.450867277,41.83728845,3],[0,0.698319762,0.715785939,0],[-2,1,-1,0],[9E+09,9E+09,9E+09,9E+09,9E+09,9E+09]];
    CONST robtarget Target_2190:=[[161.252557642,44.813302229,3],[0,0.698319762,0.715785939,0],[-2,1,-1,0],[9E+09,9E+09,9E+09,9E+09,9E+09,9E+09]];
    CONST robtarget Target_2200:=[[161.963575987,47.799477353,3],[0,0.698319762,0.715785939,0],[-2,1,-1,0],[9E+09,9E+09,9E+09,9E+09,9E+09,9E+09]];
    CONST robtarget Target_2210:=[[161.604087321,49.066373217,3],[0,0.698319762,0.715785939,0],[-2,1,-1,0],[9E+09,9E+09,9E+09,9E+09,9E+09,9E+09]];
    CONST robtarget Target_2220:=[[160.537042008,49.485484483,3],[0,0.698319762,0.715785939,0],[-2,1,-1,0],[9E+09,9E+09,9E+09,9E+09,9E+09,9E+09]];
    CONST robtarget Target_2230:=[[159.178401202,48.948082705,3],[0,0.698319762,0.715785939,0],[-2,1,-1,0],[9E+09,9E+09,9E+09,9E+09,9E+09,9E+09]];
    CONST robtarget Target_2240:=[[158.199861844,47.346320771,3],[0,0.698319762,0.715785939,0],[-2,1,-1,0],[9E+09,9E+09,9E+09,9E+09,9E+09,9E+09]];
    CONST robtarget Target_2250:=[[159.483453615,33.270063232,3],[0,0.698319762,0.715785939,0],[-2,1,-1,0],[9E+09,9E+09,9E+09,9E+09,9E+09,9E+09]];
    CONST robtarget Target_2260:=[[158.137096378,31.191079575,3],[0,0.698319762,0.715785939,0],[-2,1,-1,0],[9E+09,9E+09,9E+09,9E+09,9E+09,9E+09]];
    CONST robtarget Target_2270:=[[157.694231755,28.745724827,3],[0,0.698319762,0.715785939,0],[-2,1,-1,0],[9E+09,9E+09,9E+09,9E+09,9E+09,9E+09]];
    CONST robtarget Target_2280:=[[158.35434369,25.760644108,3],[0,0.698319762,0.715785939,0],[-2,1,-1,0],[9E+09,9E+09,9E+09,9E+09,9E+09,9E+09]];
    CONST robtarget Target_2290:=[[160.312221666,23.454800976,3],[0,0.698319762,0.715785939,0],[-2,0,-1,0],[9E+09,9E+09,9E+09,9E+09,9E+09,9E+09]];
    CONST robtarget Target_2300:=[[162.88837865,22.142087396,3],[0,0.698319762,0.715785939,0],[-2,0,-1,0],[9E+09,9E+09,9E+09,9E+09,9E+09,9E+09]];
    CONST robtarget Target_2310:=[[165.944655954,21.711925677,3],[0,0.698319762,0.715785939,0],[-2,0,-1,0],[9E+09,9E+09,9E+09,9E+09,9E+09,9E+09]];
    CONST robtarget Target_2320:=[[168.724666389,22.09783083,3],[0,0.698319762,0.715785939,0],[-2,0,-1,0],[9E+09,9E+09,9E+09,9E+09,9E+09,9E+09]];
    CONST robtarget Target_2330:=[[171.01194241,23.235138306,3],[0,0.698319762,0.715785939,0],[-2,0,-1,0],[9E+09,9E+09,9E+09,9E+09,9E+09,9E+09]];
    CONST robtarget Target_2340:=[[172.71030534,25.208725568,3],[0,0.698319762,0.715785939,0],[-2,0,-1,0],[9E+09,9E+09,9E+09,9E+09,9E+09,9E+09]];
    CONST robtarget Target_2350:=[[173.270035711,27.76101945,3],[0,0.698319762,0.715785939,0],[-2,0,-1,0],[9E+09,9E+09,9E+09,9E+09,9E+09,9E+09]];
    CONST robtarget Target_2360:=[[172.533861708,31.186329309,3],[0,0.698319762,0.715785939,0],[-2,0,-1,0],[9E+09,9E+09,9E+09,9E+09,9E+09,9E+09]];
    CONST robtarget Target_2370:=[[170.351276015,33.761382457,3],[0,0.698319762,0.715785939,0],[-2,0,-1,0],[9E+09,9E+09,9E+09,9E+09,9E+09,9E+09]];
    CONST robtarget Target_2380:=[[167.718230095,35.091642669,3],[0,0.698319762,0.715785939,0],[-2,0,-1,0],[9E+09,9E+09,9E+09,9E+09,9E+09,9E+09]];
    CONST robtarget Target_2390:=[[164.747414394,35.461705537,3],[0,0.698319762,0.715785939,0],[-2,0,-1,0],[9E+09,9E+09,9E+09,9E+09,9E+09,9E+09]];
    CONST robtarget Target_2400:=[[161.783418321,34.858523079,3],[0,0.698319762,0.715785939,0],[-2,1,-1,0],[9E+09,9E+09,9E+09,9E+09,9E+09,9E+09]];
    CONST robtarget Target_2410:=[[159.483453615,33.270063232,3],[0,0.698319762,0.715785939,0],[-2,1,-1,0],[9E+09,9E+09,9E+09,9E+09,9E+09,9E+09]];
    CONST robtarget Target_2420:=[[164.760684386,31.525990298,3],[0,0.698319762,0.715785939,0],[-2,0,-1,0],[9E+09,9E+09,9E+09,9E+09,9E+09,9E+09]];
    CONST robtarget Target_2430:=[[167.91779943,30.684159852,3],[0,0.698319762,0.715785939,0],[-2,0,-1,0],[9E+09,9E+09,9E+09,9E+09,9E+09,9E+09]];
    CONST robtarget Target_2440:=[[169.122425911,29.494710355,3],[0,0.698319762,0.715785939,0],[-2,0,-1,0],[9E+09,9E+09,9E+09,9E+09,9E+09,9E+09]];
    CONST robtarget Target_2450:=[[169.518423365,27.933078886,3],[0,0.698319762,0.715785939,0],[-2,0,-1,0],[9E+09,9E+09,9E+09,9E+09,9E+09,9E+09]];
    CONST robtarget Target_2460:=[[168.370381048,26.035943961,3],[0,0.698319762,0.715785939,0],[-2,0,-1,0],[9E+09,9E+09,9E+09,9E+09,9E+09,9E+09]];
    CONST robtarget Target_2470:=[[164.937235801,25.516419575,3],[0,0.698319762,0.715785939,0],[-2,0,-1,0],[9E+09,9E+09,9E+09,9E+09,9E+09,9E+09]];
    CONST robtarget Target_2480:=[[163.433657479,25.823928053,3],[0,0.698319762,0.715785939,0],[-2,0,-1,0],[9E+09,9E+09,9E+09,9E+09,9E+09,9E+09]];
    CONST robtarget Target_2490:=[[162.276549013,26.615700727,3],[0,0.698319762,0.715785939,0],[-2,0,-1,0],[9E+09,9E+09,9E+09,9E+09,9E+09,9E+09]];
    CONST robtarget Target_2500:=[[161.431021199,28.758324104,3],[0,0.698319762,0.715785939,0],[-2,0,-1,0],[9E+09,9E+09,9E+09,9E+09,9E+09,9E+09]];
    CONST robtarget Target_2510:=[[162.149611225,30.551032713,3],[0,0.698319762,0.715785939,0],[-2,0,-1,0],[9E+09,9E+09,9E+09,9E+09,9E+09,9E+09]];
    CONST robtarget Target_2520:=[[163.255426734,31.279367039,3],[0,0.698319762,0.715785939,0],[-2,0,-1,0],[9E+09,9E+09,9E+09,9E+09,9E+09,9E+09]];
    CONST robtarget Target_2530:=[[164.760684386,31.525990298,3],[0,0.698319762,0.715785939,0],[-2,0,-1,0],[9E+09,9E+09,9E+09,9E+09,9E+09,9E+09]];
    CONST robtarget Target_2540:=[[165.773362172,19.608522455,3],[0,0.698319762,0.715785939,0],[-2,0,-1,0],[9E+09,9E+09,9E+09,9E+09,9E+09,9E+09]];
    CONST robtarget Target_2550:=[[159.464450969,19.61567045,3],[0,0.698319762,0.715785939,0],[-2,0,-1,0],[9E+09,9E+09,9E+09,9E+09,9E+09,9E+09]];
    CONST robtarget Target_2560:=[[158.09898697,19.056940461,3],[0,0.698319762,0.715785939,0],[-2,0,-1,0],[9E+09,9E+09,9E+09,9E+09,9E+09,9E+09]];
    CONST robtarget Target_2570:=[[157.56114928,17.648487576,3],[0,0.698319762,0.715785939,0],[-2,0,-1,0],[9E+09,9E+09,9E+09,9E+09,9E+09,9E+09]];
    CONST robtarget Target_2580:=[[158.111824709,16.236571291,3],[0,0.698319762,0.715785939,0],[-2,0,-1,0],[9E+09,9E+09,9E+09,9E+09,9E+09,9E+09]];
    CONST robtarget Target_2590:=[[160.000638211,15.658639273,3],[0,0.698319762,0.715785939,0],[-2,0,-1,0],[9E+09,9E+09,9E+09,9E+09,9E+09,9E+09]];
    CONST robtarget Target_2600:=[[164.512525052,15.313742466,3],[0,0.698319762,0.715785939,0],[-2,0,-1,0],[9E+09,9E+09,9E+09,9E+09,9E+09,9E+09]];
    CONST robtarget Target_2610:=[[168.48537356,13.49504259,3],[0,0.698319762,0.715785939,0],[-2,0,-1,0],[9E+09,9E+09,9E+09,9E+09,9E+09,9E+09]];
    CONST robtarget Target_2620:=[[169.662954453,12.316679031,3],[0,0.698319762,0.715785939,0],[-2,0,-1,0],[9E+09,9E+09,9E+09,9E+09,9E+09,9E+09]];
    CONST robtarget Target_2630:=[[170.058223454,11.112522419,3],[0,0.698319762,0.715785939,0],[-2,0,-1,0],[9E+09,9E+09,9E+09,9E+09,9E+09,9E+09]];
    CONST robtarget Target_2640:=[[160.772316062,10.25669991,3],[0,0.698319762,0.715785939,0],[-2,0,-1,0],[9E+09,9E+09,9E+09,9E+09,9E+09,9E+09]];
    CONST robtarget Target_2650:=[[158.018554627,9.462384082,3],[0,0.698319762,0.715785939,0],[-2,0,-1,0],[9E+09,9E+09,9E+09,9E+09,9E+09,9E+09]];
    CONST robtarget Target_2660:=[[157.72736611,7.330137882,3],[0,0.698319762,0.715785939,0],[-2,0,-1,0],[9E+09,9E+09,9E+09,9E+09,9E+09,9E+09]];
    CONST robtarget Target_2670:=[[158.718433046,6.271404472,3],[0,0.698319762,0.715785939,0],[-2,0,-1,0],[9E+09,9E+09,9E+09,9E+09,9E+09,9E+09]];
    CONST robtarget Target_2680:=[[169.699338907,6.933584769,3],[0,0.698319762,0.715785939,0],[-2,0,-1,0],[9E+09,9E+09,9E+09,9E+09,9E+09,9E+09]];
    CONST robtarget Target_2690:=[[171.576666229,7.451430189,3],[0,0.698319762,0.715785939,0],[-2,0,0,0],[9E+09,9E+09,9E+09,9E+09,9E+09,9E+09]];
    CONST robtarget Target_2700:=[[173.255508654,8.895697527,3],[0,0.698319762,0.715785939,0],[-2,0,0,0],[9E+09,9E+09,9E+09,9E+09,9E+09,9E+09]];
    CONST robtarget Target_2710:=[[173.809080312,11.167359918,3],[0,0.698319762,0.715785939,0],[-2,0,0,0],[9E+09,9E+09,9E+09,9E+09,9E+09,9E+09]];
    CONST robtarget Target_2720:=[[173.279358428,13.410497817,3],[0,0.698319762,0.715785939,0],[-2,0,0,0],[9E+09,9E+09,9E+09,9E+09,9E+09,9E+09]];
    CONST robtarget Target_2730:=[[171.861943988,15.551192973,3],[0,0.698319762,0.715785939,0],[-2,0,-1,0],[9E+09,9E+09,9E+09,9E+09,9E+09,9E+09]];
    CONST robtarget Target_2740:=[[173.533072962,16.118087093,3],[0,0.698319762,0.715785939,0],[-2,0,0,0],[9E+09,9E+09,9E+09,9E+09,9E+09,9E+09]];
    CONST robtarget Target_2750:=[[174.085935462,17.547876768,3],[0,0.698319762,0.715785939,0],[-2,0,0,0],[9E+09,9E+09,9E+09,9E+09,9E+09,9E+09]];
    CONST robtarget Target_2760:=[[173.553026884,18.959852957,3],[0,0.698319762,0.715785939,0],[-2,0,0,0],[9E+09,9E+09,9E+09,9E+09,9E+09,9E+09]];
    CONST robtarget Target_2770:=[[171.682738774,19.516523157,3],[0,0.698319762,0.715785939,0],[-2,0,-1,0],[9E+09,9E+09,9E+09,9E+09,9E+09,9E+09]];
    CONST robtarget Target_2780:=[[165.773362172,19.608522455,3],[0,0.698319762,0.715785939,0],[-2,0,-1,0],[9E+09,9E+09,9E+09,9E+09,9E+09,9E+09]];
    CONST robtarget LiftPoint_Johnson:=[[164.402,58.247,23],[0,0.698319762,0.715785939,0],[-2,0,0,0],[9E+09,9E+09,9E+09,9E+09,9E+09,9E+09]];
    CONST robtarget Target_2790:=[[131.042928834,145.612887778,3],[0,0.698319762,0.715785939,0],[0,0,0,0],[9E+09,9E+09,9E+09,9E+09,9E+09,9E+09]];
    CONST robtarget Target_2800:=[[129.098522194,144.981156636,3],[0,0.698319762,0.715785939,0],[-1,0,1,0],[9E+09,9E+09,9E+09,9E+09,9E+09,9E+09]];
    CONST robtarget Target_2810:=[[127.670090411,143.015570106,3],[0,0.698319762,0.715785939,0],[-1,0,1,0],[9E+09,9E+09,9E+09,9E+09,9E+09,9E+09]];
    CONST robtarget Target_2820:=[[126.76138921,138.607883933,3],[0,0.698319762,0.715785939,0],[-1,0,1,0],[9E+09,9E+09,9E+09,9E+09,9E+09,9E+09]];
    CONST robtarget Target_2830:=[[126.292545841,134.386384745,3],[0,0.698319762,0.715785939,0],[-1,0,1,0],[9E+09,9E+09,9E+09,9E+09,9E+09,9E+09]];
    CONST robtarget Target_2840:=[[125.422454772,133.275189386,3],[0,0.698319762,0.715785939,0],[-1,0,1,0],[9E+09,9E+09,9E+09,9E+09,9E+09,9E+09]];
    CONST robtarget Target_2850:=[[123.938933214,132.900770036,3],[0,0.698319762,0.715785939,0],[-1,0,1,0],[9E+09,9E+09,9E+09,9E+09,9E+09,9E+09]];
    CONST robtarget Target_2860:=[[122.683049278,133.489738693,3],[0,0.698319762,0.715785939,0],[-1,0,1,0],[9E+09,9E+09,9E+09,9E+09,9E+09,9E+09]];
    CONST robtarget Target_2870:=[[121.529728163,135.265459362,3],[0,0.698319762,0.715785939,0],[-1,0,1,0],[9E+09,9E+09,9E+09,9E+09,9E+09,9E+09]];
    CONST robtarget Target_2880:=[[120.722670873,137.589378222,3],[0,0.698319762,0.715785939,0],[-1,0,1,0],[9E+09,9E+09,9E+09,9E+09,9E+09,9E+09]];
    CONST robtarget Target_2890:=[[120.44816492,139.993237194,3],[0,0.698319762,0.715785939,0],[-1,0,1,0],[9E+09,9E+09,9E+09,9E+09,9E+09,9E+09]];
    CONST robtarget Target_2900:=[[120.877155251,142.339076365,3],[0,0.698319762,0.715785939,0],[-1,0,1,0],[9E+09,9E+09,9E+09,9E+09,9E+09,9E+09]];
    CONST robtarget Target_2910:=[[123.161207235,144.435421925,3],[0,0.698319762,0.715785939,0],[-1,0,1,0],[9E+09,9E+09,9E+09,9E+09,9E+09,9E+09]];
    CONST robtarget Target_2920:=[[123.333993307,146.393222356,3],[0,0.698319762,0.715785939,0],[-1,0,1,0],[9E+09,9E+09,9E+09,9E+09,9E+09,9E+09]];
    CONST robtarget Target_2930:=[[122.222220693,147.437348494,3],[0,0.698319762,0.715785939,0],[-1,0,1,0],[9E+09,9E+09,9E+09,9E+09,9E+09,9E+09]];
    CONST robtarget Target_2940:=[[119.759854702,147.127120703,3],[0,0.698319762,0.715785939,0],[-1,0,1,0],[9E+09,9E+09,9E+09,9E+09,9E+09,9E+09]];
    CONST robtarget Target_2950:=[[118.325683573,145.811552468,3],[0,0.698319762,0.715785939,0],[-1,0,1,0],[9E+09,9E+09,9E+09,9E+09,9E+09,9E+09]];
    CONST robtarget Target_2960:=[[117.129811738,143.349453757,3],[0,0.698319762,0.715785939,0],[-1,0,1,0],[9E+09,9E+09,9E+09,9E+09,9E+09,9E+09]];
    CONST robtarget Target_2970:=[[116.739306216,140.122816067,3],[0,0.698319762,0.715785939,0],[-1,0,1,0],[9E+09,9E+09,9E+09,9E+09,9E+09,9E+09]];
    CONST robtarget Target_2980:=[[117.111106862,136.259368358,3],[0,0.698319762,0.715785939,0],[-1,0,1,0],[9E+09,9E+09,9E+09,9E+09,9E+09,9E+09]];
    CONST robtarget Target_2990:=[[118.198876862,132.853001486,3],[0,0.698319762,0.715785939,0],[-1,0,1,0],[9E+09,9E+09,9E+09,9E+09,9E+09,9E+09]];
    CONST robtarget Target_3000:=[[120.54316329,129.72793423,3],[0,0.698319762,0.715785939,0],[-1,0,1,0],[9E+09,9E+09,9E+09,9E+09,9E+09,9E+09]];
    CONST robtarget Target_3010:=[[123.768406785,128.694486507,3],[0,0.698319762,0.715785939,0],[-1,0,1,0],[9E+09,9E+09,9E+09,9E+09,9E+09,9E+09]];
    CONST robtarget Target_3020:=[[126.452085146,129.207936238,3],[0,0.698319762,0.715785939,0],[-1,0,1,0],[9E+09,9E+09,9E+09,9E+09,9E+09,9E+09]];
    CONST robtarget Target_3030:=[[128.47877474,130.727973236,3],[0,0.698319762,0.715785939,0],[-1,0,1,0],[9E+09,9E+09,9E+09,9E+09,9E+09,9E+09]];
    CONST robtarget Target_3040:=[[129.682735935,132.89526913,3],[0,0.698319762,0.715785939,0],[-1,0,1,0],[9E+09,9E+09,9E+09,9E+09,9E+09,9E+09]];
    CONST robtarget Target_3050:=[[130.909636771,140.902328578,3],[0,0.698319762,0.715785939,0],[-1,0,1,0],[9E+09,9E+09,9E+09,9E+09,9E+09,9E+09]];
    CONST robtarget Target_3060:=[[131.795906527,141.423927842,3],[0,0.698319762,0.715785939,0],[-1,0,1,0],[9E+09,9E+09,9E+09,9E+09,9E+09,9E+09]];
    CONST robtarget Target_3070:=[[132.795472653,141.001041369,3],[0,0.698319762,0.715785939,0],[-1,0,1,0],[9E+09,9E+09,9E+09,9E+09,9E+09,9E+09]];
    CONST robtarget Target_3080:=[[134.379069716,138.033260336,3],[0,0.698319762,0.715785939,0],[-1,0,1,0],[9E+09,9E+09,9E+09,9E+09,9E+09,9E+09]];
    CONST robtarget Target_3090:=[[134.544244655,135.403468403,3],[0,0.698319762,0.715785939,0],[-1,0,1,0],[9E+09,9E+09,9E+09,9E+09,9E+09,9E+09]];
    CONST robtarget Target_3100:=[[134.220187026,131.425788772,3],[0,0.698319762,0.715785939,0],[-1,0,1,0],[9E+09,9E+09,9E+09,9E+09,9E+09,9E+09]];
    CONST robtarget Target_3110:=[[135.31415443,130.39580766,3],[0,0.698319762,0.715785939,0],[-1,0,1,0],[9E+09,9E+09,9E+09,9E+09,9E+09,9E+09]];
    CONST robtarget Target_3120:=[[136.985482207,130.909396521,3],[0,0.698319762,0.715785939,0],[-1,0,1,0],[9E+09,9E+09,9E+09,9E+09,9E+09,9E+09]];
    CONST robtarget Target_3130:=[[138.308297496,134.703970649,3],[0,0.698319762,0.715785939,0],[-1,0,1,0],[9E+09,9E+09,9E+09,9E+09,9E+09,9E+09]];
    CONST robtarget Target_3140:=[[138.462886716,136.260315462,3],[0,0.698319762,0.715785939,0],[-1,0,1,0],[9E+09,9E+09,9E+09,9E+09,9E+09,9E+09]];
    CONST robtarget Target_3150:=[[137.874358409,139.618631221,3],[0,0.698319762,0.715785939,0],[-1,0,1,0],[9E+09,9E+09,9E+09,9E+09,9E+09,9E+09]];
    CONST robtarget Target_3160:=[[136.132381765,142.674684904,3],[0,0.698319762,0.715785939,0],[-1,0,1,0],[9E+09,9E+09,9E+09,9E+09,9E+09,9E+09]];
    CONST robtarget Target_3170:=[[133.700677687,144.861689825,3],[0,0.698319762,0.715785939,0],[-1,0,1,0],[9E+09,9E+09,9E+09,9E+09,9E+09,9E+09]];
    CONST robtarget Target_3180:=[[131.042928834,145.612887778,3],[0,0.698319762,0.715785939,0],[-1,0,1,0],[9E+09,9E+09,9E+09,9E+09,9E+09,9E+09]];
    CONST robtarget Target_3190:=[[131.003698009,127.752708688,3],[0,0.698319762,0.715785939,0],[0,0,0,0],[9E+09,9E+09,9E+09,9E+09,9E+09,9E+09]];
    CONST robtarget Target_3200:=[[129.721124027,127.302596197,3],[0,0.698319762,0.715785939,0],[-1,0,1,0],[9E+09,9E+09,9E+09,9E+09,9E+09,9E+09]];
    CONST robtarget Target_3210:=[[129.020458772,124.405253101,3],[0,0.698319762,0.715785939,0],[-1,0,1,0],[9E+09,9E+09,9E+09,9E+09,9E+09,9E+09]];
    CONST robtarget Target_3220:=[[128.944272005,123.298508381,3],[0,0.698319762,0.715785939,0],[-1,0,1,0],[9E+09,9E+09,9E+09,9E+09,9E+09,9E+09]];
    CONST robtarget Target_3230:=[[117.813177726,122.934189939,3],[0,0.698319762,0.715785939,0],[-1,0,1,0],[9E+09,9E+09,9E+09,9E+09,9E+09,9E+09]];
    CONST robtarget Target_3240:=[[116.879111896,121.840536394,3],[0,0.698319762,0.715785939,0],[-1,0,1,0],[9E+09,9E+09,9E+09,9E+09,9E+09,9E+09]];
    CONST robtarget Target_3250:=[[117.582974207,119.569556449,3],[0,0.698319762,0.715785939,0],[-1,0,0,0],[9E+09,9E+09,9E+09,9E+09,9E+09,9E+09]];
    CONST robtarget Target_3260:=[[121.541635199,119.09626011,3],[0,0.698319762,0.715785939,0],[-1,0,0,0],[9E+09,9E+09,9E+09,9E+09,9E+09,9E+09]];
    CONST robtarget Target_3270:=[[129.042752021,119.377309346,3],[0,0.698319762,0.715785939,0],[-1,0,0,0],[9E+09,9E+09,9E+09,9E+09,9E+09,9E+09]];
    CONST robtarget Target_3280:=[[129.26069925,115.843688015,3],[0,0.698319762,0.715785939,0],[-1,0,0,0],[9E+09,9E+09,9E+09,9E+09,9E+09,9E+09]];
    CONST robtarget Target_3290:=[[130.276558926,114.802795715,3],[0,0.698319762,0.715785939,0],[-1,0,0,0],[9E+09,9E+09,9E+09,9E+09,9E+09,9E+09]];
    CONST robtarget Target_3300:=[[132.119586192,114.954636718,3],[0,0.698319762,0.715785939,0],[-1,0,0,0],[9E+09,9E+09,9E+09,9E+09,9E+09,9E+09]];
    CONST robtarget Target_3310:=[[132.905942867,116.665862535,3],[0,0.698319762,0.715785939,0],[-1,0,0,0],[9E+09,9E+09,9E+09,9E+09,9E+09,9E+09]];
    CONST robtarget Target_3320:=[[132.821873497,119.475300785,3],[0,0.698319762,0.715785939,0],[-1,0,0,0],[9E+09,9E+09,9E+09,9E+09,9E+09,9E+09]];
    CONST robtarget Target_3330:=[[136.638667975,119.985466112,3],[0,0.698319762,0.715785939,0],[-1,0,0,0],[9E+09,9E+09,9E+09,9E+09,9E+09,9E+09]];
    CONST robtarget Target_3340:=[[137.517821102,121.565568668,3],[0,0.698319762,0.715785939,0],[-1,0,1,0],[9E+09,9E+09,9E+09,9E+09,9E+09,9E+09]];
    CONST robtarget Target_3350:=[[136.987377969,122.970419646,3],[0,0.698319762,0.715785939,0],[-1,0,1,0],[9E+09,9E+09,9E+09,9E+09,9E+09,9E+09]];
    CONST robtarget Target_3360:=[[135.664048355,123.548503526,3],[0,0.698319762,0.715785939,0],[-1,0,1,0],[9E+09,9E+09,9E+09,9E+09,9E+09,9E+09]];
    CONST robtarget Target_3370:=[[132.751764903,123.410805308,3],[0,0.698319762,0.715785939,0],[-1,0,1,0],[9E+09,9E+09,9E+09,9E+09,9E+09,9E+09]];
    CONST robtarget Target_3380:=[[132.772977002,126.600678056,3],[0,0.698319762,0.715785939,0],[-1,0,1,0],[9E+09,9E+09,9E+09,9E+09,9E+09,9E+09]];
    CONST robtarget Target_3390:=[[131.739431845,127.620205521,3],[0,0.698319762,0.715785939,0],[-1,0,1,0],[9E+09,9E+09,9E+09,9E+09,9E+09,9E+09]];
    CONST robtarget Target_3400:=[[131.003698009,127.752708688,3],[0,0.698319762,0.715785939,0],[-1,0,1,0],[9E+09,9E+09,9E+09,9E+09,9E+09,9E+09]];
    CONST robtarget Target_3410:=[[127.532213599,112.267979356,3],[0,0.698319762,0.715785939,0],[0,0,0,0],[9E+09,9E+09,9E+09,9E+09,9E+09,9E+09]];
    CONST robtarget Target_3420:=[[118.412582256,112.141319261,3],[0,0.698319762,0.715785939,0],[-1,1,-1,0],[9E+09,9E+09,9E+09,9E+09,9E+09,9E+09]];
    CONST robtarget Target_3430:=[[117.410840943,111.093624245,3],[0,0.698319762,0.715785939,0],[-1,1,-1,0],[9E+09,9E+09,9E+09,9E+09,9E+09,9E+09]];
    CONST robtarget Target_3440:=[[117.416105736,109.537808873,3],[0,0.698319762,0.715785939,0],[-1,1,-1,0],[9E+09,9E+09,9E+09,9E+09,9E+09,9E+09]];
    CONST robtarget Target_3450:=[[118.424851041,108.496892585,3],[0,0.698319762,0.715785939,0],[-1,1,-1,0],[9E+09,9E+09,9E+09,9E+09,9E+09,9E+09]];
    CONST robtarget Target_3460:=[[131.465160284,108.356151709,3],[0,0.698319762,0.715785939,0],[-1,1,-1,0],[9E+09,9E+09,9E+09,9E+09,9E+09,9E+09]];
    CONST robtarget Target_3470:=[[132.466863451,109.403846596,3],[0,0.698319762,0.715785939,0],[-1,1,-1,0],[9E+09,9E+09,9E+09,9E+09,9E+09,9E+09]];
    CONST robtarget Target_3480:=[[132.461617731,110.959662032,3],[0,0.698319762,0.715785939,0],[-1,1,-1,0],[9E+09,9E+09,9E+09,9E+09,9E+09,9E+09]];
    CONST robtarget Target_3490:=[[131.452891499,112.000578385,3],[0,0.698319762,0.715785939,0],[-1,1,-1,0],[9E+09,9E+09,9E+09,9E+09,9E+09,9E+09]];
    CONST robtarget Target_3500:=[[127.532213599,112.267979356,3],[0,0.698319762,0.715785939,0],[-1,1,-1,0],[9E+09,9E+09,9E+09,9E+09,9E+09,9E+09]];
    CONST robtarget Target_3510:=[[138.376493552,111.309950255,3],[0,0.698319762,0.715785939,0],[0,0,0,0],[9E+09,9E+09,9E+09,9E+09,9E+09,9E+09]];
    CONST robtarget Target_3520:=[[136.882379582,111.972707735,3],[0,0.698319762,0.715785939,0],[-1,1,-1,0],[9E+09,9E+09,9E+09,9E+09,9E+09,9E+09]];
    CONST robtarget Target_3530:=[[135.392749678,111.29989001,3],[0,0.698319762,0.715785939,0],[-1,1,-1,0],[9E+09,9E+09,9E+09,9E+09,9E+09,9E+09]];
    CONST robtarget Target_3540:=[[134.78710879,109.720709651,3],[0,0.698319762,0.715785939,0],[-1,1,-1,0],[9E+09,9E+09,9E+09,9E+09,9E+09,9E+09]];
    CONST robtarget Target_3550:=[[135.403360829,108.152754044,3],[0,0.698319762,0.715785939,0],[-1,1,-1,0],[9E+09,9E+09,9E+09,9E+09,9E+09,9E+09]];
    CONST robtarget Target_3560:=[[136.897469949,107.497091925,3],[0,0.698319762,0.715785939,0],[-1,1,-1,0],[9E+09,9E+09,9E+09,9E+09,9E+09,9E+09]];
    CONST robtarget Target_3570:=[[138.387104703,108.162814289,3],[0,0.698319762,0.715785939,0],[-1,1,-1,0],[9E+09,9E+09,9E+09,9E+09,9E+09,9E+09]];
    CONST robtarget Target_3580:=[[138.992769546,109.734889815,3],[0,0.698319762,0.715785939,0],[-1,1,-1,0],[9E+09,9E+09,9E+09,9E+09,9E+09,9E+09]];
    CONST robtarget Target_3590:=[[138.376493552,111.309950255,3],[0,0.698319762,0.715785939,0],[-1,1,-1,0],[9E+09,9E+09,9E+09,9E+09,9E+09,9E+09]];
    CONST robtarget Target_3600:=[[121.070177029,105.241413735,3],[0,0.698319762,0.715785939,0],[-2,0,0,0],[9E+09,9E+09,9E+09,9E+09,9E+09,9E+09]];
    CONST robtarget Target_3610:=[[117.871640784,104.921589359,3],[0,0.698319762,0.715785939,0],[-2,0,0,0],[9E+09,9E+09,9E+09,9E+09,9E+09,9E+09]];
    CONST robtarget Target_3620:=[[116.855098529,103.873844439,3],[0,0.698319762,0.715785939,0],[-2,0,0,0],[9E+09,9E+09,9E+09,9E+09,9E+09,9E+09]];
    CONST robtarget Target_3630:=[[116.861170385,102.316257944,3],[0,0.698319762,0.715785939,0],[-2,0,0,0],[9E+09,9E+09,9E+09,9E+09,9E+09,9E+09]];
    CONST robtarget Target_3640:=[[117.891008649,101.264750635,3],[0,0.698319762,0.715785939,0],[-2,0,0,0],[9E+09,9E+09,9E+09,9E+09,9E+09,9E+09]];
    CONST robtarget Target_3650:=[[123.673437696,100.760753284,3],[0,0.698319762,0.715785939,0],[-2,0,0,0],[9E+09,9E+09,9E+09,9E+09,9E+09,9E+09]];
    CONST robtarget Target_3660:=[[127.646286269,98.942034334,3],[0,0.698319762,0.715785939,0],[-2,0,0,0],[9E+09,9E+09,9E+09,9E+09,9E+09,9E+09]];
    CONST robtarget Target_3670:=[[128.823876698,97.763670807,3],[0,0.698319762,0.715785939,0],[-2,0,0,0],[9E+09,9E+09,9E+09,9E+09,9E+09,9E+09]];
    CONST robtarget Target_3680:=[[129.219136066,96.559542773,3],[0,0.698319762,0.715785939,0],[-2,0,0,0],[9E+09,9E+09,9E+09,9E+09,9E+09,9E+09]];
    CONST robtarget Target_3690:=[[119.93325738,95.703691751,3],[0,0.698319762,0.715785939,0],[-2,0,0,0],[9E+09,9E+09,9E+09,9E+09,9E+09,9E+09]];
    CONST robtarget Target_3700:=[[117.17947684,94.909385395,3],[0,0.698319762,0.715785939,0],[-2,0,0,0],[9E+09,9E+09,9E+09,9E+09,9E+09,9E+09]];
    CONST robtarget Target_3710:=[[116.888278754,92.7771487,3],[0,0.698319762,0.715785939,0],[-2,0,0,0],[9E+09,9E+09,9E+09,9E+09,9E+09,9E+09]];
    CONST robtarget Target_3720:=[[117.879345755,91.718396216,3],[0,0.698319762,0.715785939,0],[-2,0,0,0],[9E+09,9E+09,9E+09,9E+09,9E+09,9E+09]];
    CONST robtarget Target_3730:=[[128.860261088,92.380595619,3],[0,0.698319762,0.715785939,0],[-2,0,0,0],[9E+09,9E+09,9E+09,9E+09,9E+09,9E+09]];
    CONST robtarget Target_3740:=[[130.737588442,92.898431502,3],[0,0.698319762,0.715785939,0],[-2,0,0,0],[9E+09,9E+09,9E+09,9E+09,9E+09,9E+09]];
    CONST robtarget Target_3750:=[[132.41642133,94.342698808,3],[0,0.698319762,0.715785939,0],[-2,0,0,0],[9E+09,9E+09,9E+09,9E+09,9E+09,9E+09]];
    CONST robtarget Target_3760:=[[132.970002493,96.614370768,3],[0,0.698319762,0.715785939,0],[-2,0,0,0],[9E+09,9E+09,9E+09,9E+09,9E+09,9E+09]];
    CONST robtarget Target_3770:=[[132.440280545,98.85752774,3],[0,0.698319762,0.715785939,0],[-2,0,0,0],[9E+09,9E+09,9E+09,9E+09,9E+09,9E+09]];
    CONST robtarget Target_3780:=[[131.022856568,100.998222864,3],[0,0.698319762,0.715785939,0],[-2,0,0,0],[9E+09,9E+09,9E+09,9E+09,9E+09,9E+09]];
    CONST robtarget Target_3790:=[[132.69400468,101.565097974,3],[0,0.698319762,0.715785939,0],[-2,0,0,0],[9E+09,9E+09,9E+09,9E+09,9E+09,9E+09]];
    CONST robtarget Target_3800:=[[133.246857578,102.994906691,3],[0,0.698319762,0.715785939,0],[-2,0,0,0],[9E+09,9E+09,9E+09,9E+09,9E+09,9E+09]];
    CONST robtarget Target_3810:=[[132.713949097,104.40685427,3],[0,0.698319762,0.715785939,0],[-2,0,0,0],[9E+09,9E+09,9E+09,9E+09,9E+09,9E+09]];
    CONST robtarget Target_3820:=[[130.84366089,104.963553081,3],[0,0.698319762,0.715785939,0],[-2,0,0,0],[9E+09,9E+09,9E+09,9E+09,9E+09,9E+09]];
    CONST robtarget Target_3830:=[[121.070177029,105.241413735,3],[0,0.698319762,0.715785939,0],[-2,0,0,0],[9E+09,9E+09,9E+09,9E+09,9E+09,9E+09]];
    CONST robtarget Target_3840:=[[124.261233612,83.669513597,3],[0,0.698319762,0.715785939,0],[-2,0,0,0],[9E+09,9E+09,9E+09,9E+09,9E+09,9E+09]];
    CONST robtarget Target_3850:=[[117.501045479,78.552973844,3],[0,0.698319762,0.715785939,0],[-2,0,0,0],[9E+09,9E+09,9E+09,9E+09,9E+09,9E+09]];
    CONST robtarget Target_3860:=[[117.373705467,76.812012216,3],[0,0.698319762,0.715785939,0],[-2,0,0,0],[9E+09,9E+09,9E+09,9E+09,9E+09,9E+09]];
    CONST robtarget Target_3870:=[[118.393424177,75.678778581,3],[0,0.698319762,0.715785939,0],[-2,0,0,0],[9E+09,9E+09,9E+09,9E+09,9E+09,9E+09]];
    CONST robtarget Target_3880:=[[122.917388464,77.683217159,3],[0,0.698319762,0.715785939,0],[-2,0,0,0],[9E+09,9E+09,9E+09,9E+09,9E+09,9E+09]];
    CONST robtarget Target_3890:=[[126.71525228,80.651380497,3],[0,0.698319762,0.715785939,0],[-2,0,0,0],[9E+09,9E+09,9E+09,9E+09,9E+09,9E+09]];
    CONST robtarget Target_3900:=[[131.273222047,76.25857376,3],[0,0.698319762,0.715785939,0],[-2,0,0,0],[9E+09,9E+09,9E+09,9E+09,9E+09,9E+09]];
    CONST robtarget Target_3910:=[[132.637168611,76.277382386,3],[0,0.698319762,0.715785939,0],[-2,0,0,0],[9E+09,9E+09,9E+09,9E+09,9E+09,9E+09]];
    CONST robtarget Target_3920:=[[133.699037645,77.396319737,3],[0,0.698319762,0.715785939,0],[-2,0,0,0],[9E+09,9E+09,9E+09,9E+09,9E+09,9E+09]];
    CONST robtarget Target_3930:=[[133.683328661,78.898808271,3],[0,0.698319762,0.715785939,0],[-2,0,0,0],[9E+09,9E+09,9E+09,9E+09,9E+09,9E+09]];
    CONST robtarget Target_3940:=[[127.764785513,85.428963663,3],[0,0.698319762,0.715785939,0],[-2,0,0,0],[9E+09,9E+09,9E+09,9E+09,9E+09,9E+09]];
    CONST robtarget Target_3950:=[[139.427603424,85.592608702,3],[0,0.698319762,0.715785939,0],[-2,0,0,0],[9E+09,9E+09,9E+09,9E+09,9E+09,9E+09]];
    CONST robtarget Target_3960:=[[140.429325664,86.640303653,3],[0,0.698319762,0.715785939,0],[-2,0,0,0],[9E+09,9E+09,9E+09,9E+09,9E+09,9E+09]];
    CONST robtarget Target_3970:=[[140.424079945,88.196119089,3],[0,0.698319762,0.715785939,0],[-2,0,0,0],[9E+09,9E+09,9E+09,9E+09,9E+09,9E+09]];
    CONST robtarget Target_3980:=[[139.415315566,89.237035313,3],[0,0.698319762,0.715785939,0],[-2,0,0,0],[9E+09,9E+09,9E+09,9E+09,9E+09,9E+09]];
    CONST robtarget Target_3990:=[[119.665991273,89.635785303,3],[0,0.698319762,0.715785939,0],[-2,0,0,0],[9E+09,9E+09,9E+09,9E+09,9E+09,9E+09]];
    CONST robtarget Target_4000:=[[117.877414576,89.128901262,3],[0,0.698319762,0.715785939,0],[-2,0,0,0],[9E+09,9E+09,9E+09,9E+09,9E+09,9E+09]];
    CONST robtarget Target_4010:=[[117.285731841,87.624364794,3],[0,0.698319762,0.715785939,0],[-2,0,0,0],[9E+09,9E+09,9E+09,9E+09,9E+09,9E+09]];
    CONST robtarget Target_4020:=[[117.830403714,86.219561791,3],[0,0.698319762,0.715785939,0],[-2,0,0,0],[9E+09,9E+09,9E+09,9E+09,9E+09,9E+09]];
    CONST robtarget Target_4030:=[[119.196266538,85.670031439,3],[0,0.698319762,0.715785939,0],[-2,0,0,0],[9E+09,9E+09,9E+09,9E+09,9E+09,9E+09]];
    CONST robtarget Target_4040:=[[122.976154518,85.540687287,3],[0,0.698319762,0.715785939,0],[-2,0,0,0],[9E+09,9E+09,9E+09,9E+09,9E+09,9E+09]];
    CONST robtarget Target_4050:=[[124.261233612,83.669513597,3],[0,0.698319762,0.715785939,0],[-2,0,0,0],[9E+09,9E+09,9E+09,9E+09,9E+09,9E+09]];
    CONST robtarget Target_4060:=[[125.139174688,71.907861426,3],[0,0.698319762,0.715785939,0],[-2,0,0,0],[9E+09,9E+09,9E+09,9E+09,9E+09,9E+09]];
    CONST robtarget Target_4070:=[[122.45377065,66.645223838,3],[0,0.698319762,0.715785939,0],[-2,0,0,0],[9E+09,9E+09,9E+09,9E+09,9E+09,9E+09]];
    CONST robtarget Target_4080:=[[120.815485438,66.870595457,3],[0,0.698319762,0.715785939,0],[-2,0,0,0],[9E+09,9E+09,9E+09,9E+09,9E+09,9E+09]];
    CONST robtarget Target_4090:=[[120.617175868,69.846590163,3],[0,0.698319762,0.715785939,0],[-2,0,0,0],[9E+09,9E+09,9E+09,9E+09,9E+09,9E+09]];
    CONST robtarget Target_4100:=[[121.328184675,72.832765254,3],[0,0.698319762,0.715785939,0],[-2,0,0,0],[9E+09,9E+09,9E+09,9E+09,9E+09,9E+09]];
    CONST robtarget Target_4110:=[[120.968705546,74.09966115,3],[0,0.698319762,0.715785939,0],[-2,0,0,0],[9E+09,9E+09,9E+09,9E+09,9E+09,9E+09]];
    CONST robtarget Target_4120:=[[119.90166977,74.518772448,3],[0,0.698319762,0.715785939,0],[-2,0,0,0],[9E+09,9E+09,9E+09,9E+09,9E+09,9E+09]];
    CONST robtarget Target_4130:=[[118.543019428,73.981370638,3],[0,0.698319762,0.715785939,0],[-2,0,0,0],[9E+09,9E+09,9E+09,9E+09,9E+09,9E+09]];
    CONST robtarget Target_4140:=[[117.5644705,72.379618209,3],[0,0.698319762,0.715785939,0],[-2,0,0,0],[9E+09,9E+09,9E+09,9E+09,9E+09,9E+09]];
    CONST robtarget Target_4150:=[[116.993572523,68.925038884,3],[0,0.698319762,0.715785939,0],[-2,0,0,0],[9E+09,9E+09,9E+09,9E+09,9E+09,9E+09]];
    CONST robtarget Target_4160:=[[117.254079541,66.464288631,3],[0,0.698319762,0.715785939,0],[-2,0,0,0],[9E+09,9E+09,9E+09,9E+09,9E+09,9E+09]];
    CONST robtarget Target_4170:=[[118.017549701,64.424395529,3],[0,0.698319762,0.715785939,0],[-2,0,0,0],[9E+09,9E+09,9E+09,9E+09,9E+09,9E+09]];
    CONST robtarget Target_4180:=[[119.582661469,62.724664885,3],[0,0.698319762,0.715785939,0],[-2,0,0,0],[9E+09,9E+09,9E+09,9E+09,9E+09,9E+09]];
    CONST robtarget Target_4190:=[[121.733594292,62.163571714,3],[0,0.698319762,0.715785939,0],[-2,0,0,0],[9E+09,9E+09,9E+09,9E+09,9E+09,9E+09]];
    CONST robtarget Target_4200:=[[123.511442018,62.684619872,3],[0,0.698319762,0.715785939,0],[-2,0,0,0],[9E+09,9E+09,9E+09,9E+09,9E+09,9E+09]];
    CONST robtarget Target_4210:=[[125.955822503,65.687311023,3],[0,0.698319762,0.715785939,0],[-2,0,0,0],[9E+09,9E+09,9E+09,9E+09,9E+09,9E+09]];
    CONST robtarget Target_4220:=[[127.935389662,69.597759063,3],[0,0.698319762,0.715785939,0],[-2,0,0,0],[9E+09,9E+09,9E+09,9E+09,9E+09,9E+09]];
    CONST robtarget Target_4230:=[[129.289871874,69.261318686,3],[0,0.698319762,0.715785939,0],[-2,0,0,0],[9E+09,9E+09,9E+09,9E+09,9E+09,9E+09]];
    CONST robtarget Target_4240:=[[129.437441453,65.528541545,3],[0,0.698319762,0.715785939,0],[-2,0,0,0],[9E+09,9E+09,9E+09,9E+09,9E+09,9E+09]];
    CONST robtarget Target_4250:=[[128.554875039,64.960777595,3],[0,0.698319762,0.715785939,0],[-2,0,0,0],[9E+09,9E+09,9E+09,9E+09,9E+09,9E+09]];
    CONST robtarget Target_4260:=[[128.263854375,63.833777163,3],[0,0.698319762,0.715785939,0],[-2,0,0,0],[9E+09,9E+09,9E+09,9E+09,9E+09,9E+09]];
    CONST robtarget Target_4270:=[[128.906717302,62.802279837,3],[0,0.698319762,0.715785939,0],[-2,0,0,0],[9E+09,9E+09,9E+09,9E+09,9E+09,9E+09]];
    CONST robtarget Target_4280:=[[130.82599327,62.464196079,3],[0,0.698319762,0.715785939,0],[-2,0,0,0],[9E+09,9E+09,9E+09,9E+09,9E+09,9E+09]];
    CONST robtarget Target_4290:=[[131.951218781,62.702423538,3],[0,0.698319762,0.715785939,0],[-2,0,0,0],[9E+09,9E+09,9E+09,9E+09,9E+09,9E+09]];
    CONST robtarget Target_4300:=[[132.929844424,64.275766107,3],[0,0.698319762,0.715785939,0],[-2,0,0,0],[9E+09,9E+09,9E+09,9E+09,9E+09,9E+09]];
    CONST robtarget Target_4310:=[[132.861726515,68.673058608,3],[0,0.698319762,0.715785939,0],[-2,0,0,0],[9E+09,9E+09,9E+09,9E+09,9E+09,9E+09]];
    CONST robtarget Target_4320:=[[132.417286553,70.909388673,3],[0,0.698319762,0.715785939,0],[-2,0,0,0],[9E+09,9E+09,9E+09,9E+09,9E+09,9E+09]];
    CONST robtarget Target_4330:=[[130.949719079,73.174245956,3],[0,0.698319762,0.715785939,0],[-2,0,0,0],[9E+09,9E+09,9E+09,9E+09,9E+09,9E+09]];
    CONST robtarget Target_4340:=[[128.556625338,73.922779018,3],[0,0.698319762,0.715785939,0],[-2,0,0,0],[9E+09,9E+09,9E+09,9E+09,9E+09,9E+09]];
    CONST robtarget Target_4350:=[[126.693471701,73.415653063,3],[0,0.698319762,0.715785939,0],[-2,0,0,0],[9E+09,9E+09,9E+09,9E+09,9E+09,9E+09]];
    CONST robtarget Target_4360:=[[125.139174688,71.907861426,3],[0,0.698319762,0.715785939,0],[-2,0,0,0],[9E+09,9E+09,9E+09,9E+09,9E+09,9E+09]];
    CONST robtarget LiftPoint_stinks:=[[127.806,110.712,23],[0,0.698319762,0.715785939,0],[-1,0,0,0],[9E+09,9E+09,9E+09,9E+09,9E+09,9E+09]];
    PROC Tyler_T()
        MoveL Target_10,v30,z15,My_Mechanism_1\WObj:=Workobject_1;
        WaitTime 0.5;
        MoveL Target_20,v30,z15,My_Mechanism_1\WObj:=Workobject_1;
        MoveL Target_30,v30,z15,My_Mechanism_1\WObj:=Workobject_1;
        MoveL Target_40,v30,z15,My_Mechanism_1\WObj:=Workobject_1;
        MoveL Target_50,v30,z15,My_Mechanism_1\WObj:=Workobject_1;
        MoveL Target_60,v30,z15,My_Mechanism_1\WObj:=Workobject_1;
        MoveL Target_90,v30,z15,My_Mechanism_1\WObj:=Workobject_1;
        MoveL Target_100,v30,z15,My_Mechanism_1\WObj:=Workobject_1;
        MoveL Target_110,v30,z15,My_Mechanism_1\WObj:=Workobject_1;
        MoveL Target_120,v30,z15,My_Mechanism_1\WObj:=Workobject_1;
        MoveL Target_130,v30,z15,My_Mechanism_1\WObj:=Workobject_1;
        MoveL Target_140,v30,z15,My_Mechanism_1\WObj:=Workobject_1;
        MoveL Target_150,v30,z15,My_Mechanism_1\WObj:=Workobject_1;
        MoveL Target_160,v30,z15,My_Mechanism_1\WObj:=Workobject_1;
        WaitTime 0.5;
    ENDPROC
    PROC Tyler_y()
        MoveL Target_170,v30,z15,My_Mechanism_1\WObj:=Workobject_1;
        WaitTime 0.5;
        MoveL Target_180,v30,z15,My_Mechanism_1\WObj:=Workobject_1;
        MoveL Target_190,v30,z15,My_Mechanism_1\WObj:=Workobject_1;
        MoveL Target_200,v30,z15,My_Mechanism_1\WObj:=Workobject_1;
        MoveL Target_210,v30,z15,My_Mechanism_1\WObj:=Workobject_1;
        MoveL Target_220,v30,z15,My_Mechanism_1\WObj:=Workobject_1;
        MoveL Target_230,v30,z15,My_Mechanism_1\WObj:=Workobject_1;
        MoveL Target_240,v30,z15,My_Mechanism_1\WObj:=Workobject_1;
        MoveL Target_250,v30,z15,My_Mechanism_1\WObj:=Workobject_1;
        MoveL Target_260,v30,z15,My_Mechanism_1\WObj:=Workobject_1;
        MoveL Target_270,v30,z15,My_Mechanism_1\WObj:=Workobject_1;
        MoveL Target_280,v30,z15,My_Mechanism_1\WObj:=Workobject_1;
        MoveL Target_290,v30,z15,My_Mechanism_1\WObj:=Workobject_1;
        MoveL Target_300,v30,z15,My_Mechanism_1\WObj:=Workobject_1;
        MoveL Target_310,v30,z15,My_Mechanism_1\WObj:=Workobject_1;
        MoveL Target_320,v30,z15,My_Mechanism_1\WObj:=Workobject_1;
        WaitTime 0.5;
    ENDPROC
    PROC Tyler_l()
        MoveL Target_330,v30,z15,My_Mechanism_1\WObj:=Workobject_1;
        WaitTime 0.5;
        MoveL Target_340,v30,z15,My_Mechanism_1\WObj:=Workobject_1;
        MoveL Target_350,v30,z15,My_Mechanism_1\WObj:=Workobject_1;
        MoveL Target_360,v30,z15,My_Mechanism_1\WObj:=Workobject_1;
        MoveL Target_370,v30,z15,My_Mechanism_1\WObj:=Workobject_1;
        MoveL Target_380,v30,z15,My_Mechanism_1\WObj:=Workobject_1;
        MoveL Target_390,v30,z15,My_Mechanism_1\WObj:=Workobject_1;
        MoveL Target_400,v30,z15,My_Mechanism_1\WObj:=Workobject_1;
        MoveL Target_410,v30,z15,My_Mechanism_1\WObj:=Workobject_1;
        WaitTime 0.5;
    ENDPROC
    PROC Tyler_e()
        MoveL Target_420,v30,z15,My_Mechanism_1\WObj:=Workobject_1;
        WaitTime 0.5;
        MoveL Target_430,v30,z15,My_Mechanism_1\WObj:=Workobject_1;
        MoveL Target_440,v30,z15,My_Mechanism_1\WObj:=Workobject_1;
        MoveL Target_450,v30,z15,My_Mechanism_1\WObj:=Workobject_1;
        MoveL Target_460,v30,z15,My_Mechanism_1\WObj:=Workobject_1;
        MoveL Target_470,v30,z15,My_Mechanism_1\WObj:=Workobject_1;
        MoveL Target_480,v30,z15,My_Mechanism_1\WObj:=Workobject_1;
        MoveL Target_490,v30,z15,My_Mechanism_1\WObj:=Workobject_1;
        MoveL Target_500,v30,z15,My_Mechanism_1\WObj:=Workobject_1;
        MoveL Target_510,v30,z15,My_Mechanism_1\WObj:=Workobject_1;
        MoveL Target_520,v30,z15,My_Mechanism_1\WObj:=Workobject_1;
        MoveL Target_530,v30,z15,My_Mechanism_1\WObj:=Workobject_1;
        MoveL Target_540,v30,z15,My_Mechanism_1\WObj:=Workobject_1;
        MoveL Target_550,v30,z15,My_Mechanism_1\WObj:=Workobject_1;
        MoveL Target_560,v30,z15,My_Mechanism_1\WObj:=Workobject_1;
        MoveL Target_570,v30,z15,My_Mechanism_1\WObj:=Workobject_1;
        MoveL Target_580,v30,z15,My_Mechanism_1\WObj:=Workobject_1;
        MoveL Target_590,v30,z15,My_Mechanism_1\WObj:=Workobject_1;
        MoveL Target_600,v30,z15,My_Mechanism_1\WObj:=Workobject_1;
        MoveL Target_610,v30,z15,My_Mechanism_1\WObj:=Workobject_1;
        MoveL Target_620,v30,z15,My_Mechanism_1\WObj:=Workobject_1;
        MoveL Target_630,v30,z15,My_Mechanism_1\WObj:=Workobject_1;
        MoveL Target_640,v30,z15,My_Mechanism_1\WObj:=Workobject_1;
        WaitTime 0.5;
        MoveJ liftPoint_Tyler,v30,z15,My_Mechanism_1\WObj:=Workobject_1;
        Tyler_e_inner;
    ENDPROC
    PROC Tyler_e_inner()
        MoveL Target_650,v30,z15,My_Mechanism_1\WObj:=Workobject_1;
        WaitTime 0.5;
        MoveL Target_660,v30,z15,My_Mechanism_1\WObj:=Workobject_1;
        MoveL Target_670,v30,z15,My_Mechanism_1\WObj:=Workobject_1;
        MoveL Target_680,v30,z15,My_Mechanism_1\WObj:=Workobject_1;
        MoveL Target_690,v30,z15,My_Mechanism_1\WObj:=Workobject_1;
        WaitTime 0.5;
    ENDPROC
    PROC Tyler_r()
        MoveL Target_700,v30,z15,My_Mechanism_1\WObj:=Workobject_1;
        WaitTime 0.5;
        MoveL Target_710,v30,z15,My_Mechanism_1\WObj:=Workobject_1;
        MoveL Target_720,v30,z15,My_Mechanism_1\WObj:=Workobject_1;
        MoveL Target_730,v30,z15,My_Mechanism_1\WObj:=Workobject_1;
        MoveL Target_740,v30,z15,My_Mechanism_1\WObj:=Workobject_1;
        MoveL Target_750,v30,z15,My_Mechanism_1\WObj:=Workobject_1;
        MoveL Target_760,v30,z15,My_Mechanism_1\WObj:=Workobject_1;
        MoveL Target_770,v30,z15,My_Mechanism_1\WObj:=Workobject_1;
        MoveL Target_780,v30,z15,My_Mechanism_1\WObj:=Workobject_1;
        MoveL Target_790,v30,z15,My_Mechanism_1\WObj:=Workobject_1;
        MoveL Target_800,v30,z15,My_Mechanism_1\WObj:=Workobject_1;
        MoveL Target_810,v30,z15,My_Mechanism_1\WObj:=Workobject_1;
        MoveL Target_820,v30,z15,My_Mechanism_1\WObj:=Workobject_1;
        MoveL Target_830,v30,z15,My_Mechanism_1\WObj:=Workobject_1;
        MoveL Target_840,v30,z15,My_Mechanism_1\WObj:=Workobject_1;
        MoveL Target_850,v30,z15,My_Mechanism_1\WObj:=Workobject_1;
        MoveL Target_860,v30,z15,My_Mechanism_1\WObj:=Workobject_1;
        MoveL Target_870,v30,z15,My_Mechanism_1\WObj:=Workobject_1;
        MoveL Target_880,v30,z15,My_Mechanism_1\WObj:=Workobject_1;
        MoveL Target_890,v30,z15,My_Mechanism_1\WObj:=Workobject_1;
        WaitTime 0.5;
    ENDPROC
    PROC main()
        MoveJ Homes,v30,z15,My_Mechanism_1\WObj:=wobj0;
        MoveJ liftPoint_Tyler,v30,z15,My_Mechanism_1\WObj:=Workobject_1;
        Tyler_T;
        MoveJ liftPoint_Tyler,v30,z15,My_Mechanism_1\WObj:=Workobject_1;
        Tyler_y;
        MoveJ liftPoint_Tyler,v30,z15,My_Mechanism_1\WObj:=Workobject_1;
        Tyler_l;
        MoveJ liftPoint_Tyler,v30,z15,My_Mechanism_1\WObj:=Workobject_1;
        Tyler_e;
        MoveJ liftPoint_Tyler,v30,z15,My_Mechanism_1\WObj:=Workobject_1;
        Tyler_r;
        MoveL LiftPoint_Johnson,v30,z15,My_Mechanism_1\WObj:=Workobject_1;
        Johnson_J;
        MoveL LiftPoint_Johnson,v30,z15,My_Mechanism_1\WObj:=Workobject_1;
        Johnson_o_1;
        MoveL LiftPoint_Johnson,v30,z15,My_Mechanism_1\WObj:=Workobject_1;
        Johnson_h;
        MoveL LiftPoint_Johnson,v30,z15,My_Mechanism_1\WObj:=Workobject_1;
        Johnson_n;
        MoveL LiftPoint_Johnson,v30,z15,My_Mechanism_1\WObj:=Workobject_1;
        Johnson_s;
        MoveL LiftPoint_Johnson,v30,z15,My_Mechanism_1\WObj:=Workobject_1;
        Johnson_o_2;
        MoveL LiftPoint_Johnson,v30,z15,My_Mechanism_1\WObj:=Workobject_1;
        Johnson_n_2;
        MoveL LiftPoint_stinks,v30,z15,My_Mechanism_1\WObj:=Workobject_1;
        Stinks_S;
        MoveL LiftPoint_stinks,v30,z15,My_Mechanism_1\WObj:=Workobject_1;
        Stinks_t;
        MoveL LiftPoint_stinks,v30,z15,My_Mechanism_1\WObj:=Workobject_1;
        Stinks_i;
        MoveL LiftPoint_stinks,v30,z15,My_Mechanism_1\WObj:=Workobject_1;
        Stinks_n;
        MoveL LiftPoint_stinks,v30,z15,My_Mechanism_1\WObj:=Workobject_1;
        Stinks_k;
        MoveL LiftPoint_stinks,v30,z15,My_Mechanism_1\WObj:=Workobject_1;
        Stinks_s_2;
        MoveL LiftPoint_stinks,v30,z15,My_Mechanism_1\WObj:=Workobject_1;
        MoveJ Homes,v30,z15,My_Mechanism_1\WObj:=wobj0;
    ENDPROC
    PROC Johnson_J()
        MoveL Target_900,v30,z15,My_Mechanism_1\WObj:=Workobject_1;
        WaitTime 0.5;
        MoveL Target_910,v30,z15,My_Mechanism_1\WObj:=Workobject_1;
        MoveL Target_920,v30,z15,My_Mechanism_1\WObj:=Workobject_1;
        MoveL Target_930,v30,z15,My_Mechanism_1\WObj:=Workobject_1;
        MoveL Target_940,v30,z15,My_Mechanism_1\WObj:=Workobject_1;
        MoveL Target_950,v30,z15,My_Mechanism_1\WObj:=Workobject_1;
        MoveL Target_960,v30,z15,My_Mechanism_1\WObj:=Workobject_1;
        MoveL Target_970,v30,z15,My_Mechanism_1\WObj:=Workobject_1;
        MoveL Target_980,v30,z15,My_Mechanism_1\WObj:=Workobject_1;
        MoveL Target_990,v30,z15,My_Mechanism_1\WObj:=Workobject_1;
        MoveL Target_1000,v30,z15,My_Mechanism_1\WObj:=Workobject_1;
        MoveL Target_1010,v30,z15,My_Mechanism_1\WObj:=Workobject_1;
        MoveL Target_1020,v30,z15,My_Mechanism_1\WObj:=Workobject_1;
        MoveL Target_1030,v30,z15,My_Mechanism_1\WObj:=Workobject_1;
        MoveL Target_1040,v30,z15,My_Mechanism_1\WObj:=Workobject_1;
        MoveL Target_1050,v30,z15,My_Mechanism_1\WObj:=Workobject_1;
        MoveL Target_1060,v30,z15,My_Mechanism_1\WObj:=Workobject_1;
        MoveL Target_1070,v30,z15,My_Mechanism_1\WObj:=Workobject_1;
        MoveL Target_1080,v30,z15,My_Mechanism_1\WObj:=Workobject_1;
        MoveL Target_1090,v30,z15,My_Mechanism_1\WObj:=Workobject_1;
        MoveL Target_1100,v30,z15,My_Mechanism_1\WObj:=Workobject_1;
        MoveL Target_1110,v30,z15,My_Mechanism_1\WObj:=Workobject_1;
        MoveL Target_1120,v30,z15,My_Mechanism_1\WObj:=Workobject_1;
        MoveL Target_1130,v30,z15,My_Mechanism_1\WObj:=Workobject_1;
        MoveL Target_1140,v30,z15,My_Mechanism_1\WObj:=Workobject_1;
        MoveL Target_1150,v30,z15,My_Mechanism_1\WObj:=Workobject_1;
        MoveL Target_1160,v30,z15,My_Mechanism_1\WObj:=Workobject_1;
        WaitTime 0.5;
    ENDPROC
    PROC Johnson_o_1()
        MoveL Target_1170,v30,z15,My_Mechanism_1\WObj:=Workobject_1;
        WaitTime 0.5;
        MoveL Target_1180,v30,z15,My_Mechanism_1\WObj:=Workobject_1;
        MoveL Target_1190,v30,z15,My_Mechanism_1\WObj:=Workobject_1;
        MoveL Target_1200,v30,z15,My_Mechanism_1\WObj:=Workobject_1;
        MoveL Target_1210,v30,z15,My_Mechanism_1\WObj:=Workobject_1;
        MoveL Target_1220,v30,z15,My_Mechanism_1\WObj:=Workobject_1;
        MoveL Target_1230,v30,z15,My_Mechanism_1\WObj:=Workobject_1;
        MoveL Target_1240,v30,z15,My_Mechanism_1\WObj:=Workobject_1;
        MoveL Target_1250,v30,z15,My_Mechanism_1\WObj:=Workobject_1;
        MoveL Target_1260,v30,z15,My_Mechanism_1\WObj:=Workobject_1;
        MoveL Target_1270,v30,z15,My_Mechanism_1\WObj:=Workobject_1;
        MoveL Target_1280,v30,z15,My_Mechanism_1\WObj:=Workobject_1;
        MoveL Target_1290,v30,z15,My_Mechanism_1\WObj:=Workobject_1;
        MoveL Target_1300,v30,z15,My_Mechanism_1\WObj:=Workobject_1;
        MoveL Target_1310,v30,z15,My_Mechanism_1\WObj:=Workobject_1;
        MoveL Target_1320,v30,z15,My_Mechanism_1\WObj:=Workobject_1;
        MoveL Target_1330,v30,z15,My_Mechanism_1\WObj:=Workobject_1;
        WaitTime 0.5;
        MoveL LiftPoint_Johnson,v30,z15,My_Mechanism_1\WObj:=Workobject_1;
        Johnson_o_1_inner;
    ENDPROC
    PROC Johnson_o_1_inner()
        MoveL Target_1340,v30,z15,My_Mechanism_1\WObj:=Workobject_1;
        WaitTime 0.5;
        MoveL Target_1350,v30,z15,My_Mechanism_1\WObj:=Workobject_1;
        MoveL Target_1360,v30,z15,My_Mechanism_1\WObj:=Workobject_1;
        MoveL Target_1370,v30,z15,My_Mechanism_1\WObj:=Workobject_1;
        MoveL Target_1380,v30,z15,My_Mechanism_1\WObj:=Workobject_1;
        MoveL Target_1390,v30,z15,My_Mechanism_1\WObj:=Workobject_1;
        MoveL Target_1400,v30,z15,My_Mechanism_1\WObj:=Workobject_1;
        MoveL Target_1410,v30,z15,My_Mechanism_1\WObj:=Workobject_1;
        MoveL Target_1420,v30,z15,My_Mechanism_1\WObj:=Workobject_1;
        MoveL Target_1430,v30,z15,My_Mechanism_1\WObj:=Workobject_1;
        MoveL Target_1440,v30,z15,My_Mechanism_1\WObj:=Workobject_1;
        MoveL Target_1450,v30,z15,My_Mechanism_1\WObj:=Workobject_1;
        WaitTime 0.5;
    ENDPROC
    PROC Johnson_h()
        MoveL Target_1460,v30,z15,My_Mechanism_1\WObj:=Workobject_1;
        WaitTime 0.5;
        MoveL Target_1470,v30,z15,My_Mechanism_1\WObj:=Workobject_1;
        MoveL Target_1480,v30,z15,My_Mechanism_1\WObj:=Workobject_1;
        MoveL Target_1490,v30,z15,My_Mechanism_1\WObj:=Workobject_1;
        MoveL Target_1500,v30,z15,My_Mechanism_1\WObj:=Workobject_1;
        MoveL Target_1510,v30,z15,My_Mechanism_1\WObj:=Workobject_1;
        MoveL Target_1520,v30,z15,My_Mechanism_1\WObj:=Workobject_1;
        MoveL Target_1530,v30,z15,My_Mechanism_1\WObj:=Workobject_1;
        MoveL Target_1540,v30,z15,My_Mechanism_1\WObj:=Workobject_1;
        MoveL Target_1550,v30,z15,My_Mechanism_1\WObj:=Workobject_1;
        MoveL Target_1560,v30,z15,My_Mechanism_1\WObj:=Workobject_1;
        MoveL Target_1570,v30,z15,My_Mechanism_1\WObj:=Workobject_1;
        MoveL Target_1580,v30,z15,My_Mechanism_1\WObj:=Workobject_1;
        MoveL Target_1590,v30,z15,My_Mechanism_1\WObj:=Workobject_1;
        MoveL Target_1600,v30,z15,My_Mechanism_1\WObj:=Workobject_1;
        MoveL Target_1610,v30,z15,My_Mechanism_1\WObj:=Workobject_1;
        MoveL Target_1620,v30,z15,My_Mechanism_1\WObj:=Workobject_1;
        MoveL Target_1630,v30,z15,My_Mechanism_1\WObj:=Workobject_1;
        MoveL Target_1640,v30,z15,My_Mechanism_1\WObj:=Workobject_1;
        MoveL Target_1650,v30,z15,My_Mechanism_1\WObj:=Workobject_1;
        MoveL Target_1660,v30,z15,My_Mechanism_1\WObj:=Workobject_1;
        MoveL Target_1670,v30,z15,My_Mechanism_1\WObj:=Workobject_1;
        MoveL Target_1680,v30,z15,My_Mechanism_1\WObj:=Workobject_1;
        WaitTime 0.5;
    ENDPROC
    PROC Johnson_n()
        MoveL Target_1690,v30,z15,My_Mechanism_1\WObj:=Workobject_1;
        WaitTime 0.5;
        MoveL Target_1700,v30,z15,My_Mechanism_1\WObj:=Workobject_1;
        MoveL Target_1710,v30,z15,My_Mechanism_1\WObj:=Workobject_1;
        MoveL Target_1720,v30,z15,My_Mechanism_1\WObj:=Workobject_1;
        MoveL Target_1730,v30,z15,My_Mechanism_1\WObj:=Workobject_1;
        MoveL Target_1740,v30,z15,My_Mechanism_1\WObj:=Workobject_1;
        MoveL Target_1750,v30,z15,My_Mechanism_1\WObj:=Workobject_1;
        MoveL Target_1760,v30,z15,My_Mechanism_1\WObj:=Workobject_1;
        MoveL Target_1770,v30,z15,My_Mechanism_1\WObj:=Workobject_1;
        MoveL Target_1780,v30,z15,My_Mechanism_1\WObj:=Workobject_1;
        MoveL Target_1790,v30,z15,My_Mechanism_1\WObj:=Workobject_1;
        MoveL Target_1800,v30,z15,My_Mechanism_1\WObj:=Workobject_1;
        MoveL Target_1810,v30,z15,My_Mechanism_1\WObj:=Workobject_1;
        MoveL Target_1820,v30,z15,My_Mechanism_1\WObj:=Workobject_1;
        MoveL Target_1830,v30,z15,My_Mechanism_1\WObj:=Workobject_1;
        MoveL Target_1840,v30,z15,My_Mechanism_1\WObj:=Workobject_1;
        MoveL Target_1850,v30,z15,My_Mechanism_1\WObj:=Workobject_1;
        MoveL Target_1860,v30,z15,My_Mechanism_1\WObj:=Workobject_1;
        MoveL Target_1870,v30,z15,My_Mechanism_1\WObj:=Workobject_1;
        MoveL Target_1880,v30,z15,My_Mechanism_1\WObj:=Workobject_1;
        MoveL Target_1890,v30,z15,My_Mechanism_1\WObj:=Workobject_1;
        MoveL Target_1900,v30,z15,My_Mechanism_1\WObj:=Workobject_1;
        MoveL Target_1910,v30,z15,My_Mechanism_1\WObj:=Workobject_1;
        MoveL Target_1920,v30,z15,My_Mechanism_1\WObj:=Workobject_1;
        MoveL Target_1930,v30,z15,My_Mechanism_1\WObj:=Workobject_1;
        WaitTime 0.5;
    ENDPROC
    PROC Johnson_s()
        MoveL Target_1940,v30,z15,My_Mechanism_1\WObj:=Workobject_1;
        WaitTime 0.5;
        MoveL Target_1950,v30,z15,My_Mechanism_1\WObj:=Workobject_1;
        MoveL Target_1960,v30,z15,My_Mechanism_1\WObj:=Workobject_1;
        MoveL Target_1970,v30,z15,My_Mechanism_1\WObj:=Workobject_1;
        MoveL Target_1980,v30,z15,My_Mechanism_1\WObj:=Workobject_1;
        MoveL Target_1990,v30,z15,My_Mechanism_1\WObj:=Workobject_1;
        MoveL Target_2000,v30,z15,My_Mechanism_1\WObj:=Workobject_1;
        MoveL Target_2010,v30,z15,My_Mechanism_1\WObj:=Workobject_1;
        MoveL Target_2020,v30,z15,My_Mechanism_1\WObj:=Workobject_1;
        MoveL Target_2030,v30,z15,My_Mechanism_1\WObj:=Workobject_1;
        MoveL Target_2040,v30,z15,My_Mechanism_1\WObj:=Workobject_1;
        MoveL Target_2050,v30,z15,My_Mechanism_1\WObj:=Workobject_1;
        MoveL Target_2060,v30,z15,My_Mechanism_1\WObj:=Workobject_1;
        MoveL Target_2070,v30,z15,My_Mechanism_1\WObj:=Workobject_1;
        MoveL Target_2080,v30,z15,My_Mechanism_1\WObj:=Workobject_1;
        MoveL Target_2090,v30,z15,My_Mechanism_1\WObj:=Workobject_1;
        MoveL Target_2100,v30,z15,My_Mechanism_1\WObj:=Workobject_1;
        MoveL Target_2110,v30,z15,My_Mechanism_1\WObj:=Workobject_1;
        MoveL Target_2120,v30,z15,My_Mechanism_1\WObj:=Workobject_1;
        MoveL Target_2130,v30,z15,My_Mechanism_1\WObj:=Workobject_1;
        MoveL Target_2140,v30,z15,My_Mechanism_1\WObj:=Workobject_1;
        MoveL Target_2150,v30,z15,My_Mechanism_1\WObj:=Workobject_1;
        MoveL Target_2160,v30,z15,My_Mechanism_1\WObj:=Workobject_1;
        MoveL Target_2170,v30,z15,My_Mechanism_1\WObj:=Workobject_1;
        MoveL Target_2180,v30,z15,My_Mechanism_1\WObj:=Workobject_1;
        MoveL Target_2190,v30,z15,My_Mechanism_1\WObj:=Workobject_1;
        MoveL Target_2200,v30,z15,My_Mechanism_1\WObj:=Workobject_1;
        MoveL Target_2210,v30,z15,My_Mechanism_1\WObj:=Workobject_1;
        MoveL Target_2220,v30,z15,My_Mechanism_1\WObj:=Workobject_1;
        MoveL Target_2230,v30,z15,My_Mechanism_1\WObj:=Workobject_1;
        MoveL Target_2240,v30,z15,My_Mechanism_1\WObj:=Workobject_1;
        WaitTime 0.5;
    ENDPROC
    PROC Johnson_o_2()
        MoveL Target_2250,v30,z15,My_Mechanism_1\WObj:=Workobject_1;
        WaitTime 0.5;
        MoveL Target_2260,v30,z15,My_Mechanism_1\WObj:=Workobject_1;
        MoveL Target_2270,v30,z15,My_Mechanism_1\WObj:=Workobject_1;
        MoveL Target_2280,v30,z15,My_Mechanism_1\WObj:=Workobject_1;
        MoveL Target_2290,v30,z15,My_Mechanism_1\WObj:=Workobject_1;
        MoveL Target_2300,v30,z15,My_Mechanism_1\WObj:=Workobject_1;
        MoveL Target_2310,v30,z15,My_Mechanism_1\WObj:=Workobject_1;
        MoveL Target_2320,v30,z15,My_Mechanism_1\WObj:=Workobject_1;
        MoveL Target_2330,v30,z15,My_Mechanism_1\WObj:=Workobject_1;
        MoveL Target_2340,v30,z15,My_Mechanism_1\WObj:=Workobject_1;
        MoveL Target_2350,v30,z15,My_Mechanism_1\WObj:=Workobject_1;
        MoveL Target_2360,v30,z15,My_Mechanism_1\WObj:=Workobject_1;
        MoveL Target_2370,v30,z15,My_Mechanism_1\WObj:=Workobject_1;
        MoveL Target_2380,v30,z15,My_Mechanism_1\WObj:=Workobject_1;
        MoveL Target_2390,v30,z15,My_Mechanism_1\WObj:=Workobject_1;
        MoveL Target_2400,v30,z15,My_Mechanism_1\WObj:=Workobject_1;
        MoveL Target_2410,v30,z15,My_Mechanism_1\WObj:=Workobject_1;
        WaitTime 0.5;
        MoveL LiftPoint_Johnson,v30,z15,My_Mechanism_1\WObj:=Workobject_1;
        Johnson_o_2_inner;
    ENDPROC
    PROC Johnson_o_2_inner()
        MoveL Target_2420,v30,z15,My_Mechanism_1\WObj:=Workobject_1;
        WaitTime 0.5;
        MoveL Target_2430,v30,z15,My_Mechanism_1\WObj:=Workobject_1;
        MoveL Target_2440,v30,z15,My_Mechanism_1\WObj:=Workobject_1;
        MoveL Target_2450,v30,z15,My_Mechanism_1\WObj:=Workobject_1;
        MoveL Target_2460,v30,z15,My_Mechanism_1\WObj:=Workobject_1;
        MoveL Target_2470,v30,z15,My_Mechanism_1\WObj:=Workobject_1;
        MoveL Target_2480,v30,z15,My_Mechanism_1\WObj:=Workobject_1;
        MoveL Target_2490,v30,z15,My_Mechanism_1\WObj:=Workobject_1;
        MoveL Target_2500,v30,z15,My_Mechanism_1\WObj:=Workobject_1;
        MoveL Target_2510,v30,z15,My_Mechanism_1\WObj:=Workobject_1;
        MoveL Target_2520,v30,z15,My_Mechanism_1\WObj:=Workobject_1;
        MoveL Target_2530,v30,z15,My_Mechanism_1\WObj:=Workobject_1;
        WaitTime 0.5;
    ENDPROC
    PROC Johnson_n_2()
        MoveL Target_2540,v30,z15,My_Mechanism_1\WObj:=Workobject_1;
        WaitTime 0.5;
        MoveL Target_2550,v30,z15,My_Mechanism_1\WObj:=Workobject_1;
        MoveL Target_2560,v30,z15,My_Mechanism_1\WObj:=Workobject_1;
        MoveL Target_2570,v30,z15,My_Mechanism_1\WObj:=Workobject_1;
        MoveL Target_2580,v30,z15,My_Mechanism_1\WObj:=Workobject_1;
        MoveL Target_2590,v30,z15,My_Mechanism_1\WObj:=Workobject_1;
        MoveL Target_2600,v30,z15,My_Mechanism_1\WObj:=Workobject_1;
        MoveL Target_2610,v30,z15,My_Mechanism_1\WObj:=Workobject_1;
        MoveL Target_2620,v30,z15,My_Mechanism_1\WObj:=Workobject_1;
        MoveL Target_2630,v30,z15,My_Mechanism_1\WObj:=Workobject_1;
        MoveL Target_2640,v30,z15,My_Mechanism_1\WObj:=Workobject_1;
        MoveL Target_2650,v30,z15,My_Mechanism_1\WObj:=Workobject_1;
        MoveL Target_2660,v30,z15,My_Mechanism_1\WObj:=Workobject_1;
        MoveL Target_2670,v30,z15,My_Mechanism_1\WObj:=Workobject_1;
        MoveL Target_2680,v30,z15,My_Mechanism_1\WObj:=Workobject_1;
        MoveL Target_2690,v30,z15,My_Mechanism_1\WObj:=Workobject_1;
        MoveL Target_2700,v30,z15,My_Mechanism_1\WObj:=Workobject_1;
        MoveL Target_2710,v30,z15,My_Mechanism_1\WObj:=Workobject_1;
        MoveL Target_2720,v30,z15,My_Mechanism_1\WObj:=Workobject_1;
        MoveL Target_2730,v30,z15,My_Mechanism_1\WObj:=Workobject_1;
        MoveL Target_2740,v30,z15,My_Mechanism_1\WObj:=Workobject_1;
        MoveL Target_2750,v30,z15,My_Mechanism_1\WObj:=Workobject_1;
        MoveL Target_2760,v30,z15,My_Mechanism_1\WObj:=Workobject_1;
        MoveL Target_2770,v30,z15,My_Mechanism_1\WObj:=Workobject_1;
        MoveL Target_2780,v30,z15,My_Mechanism_1\WObj:=Workobject_1;
        WaitTime 0.5;
    ENDPROC
    PROC Stinks_S()
        MoveL Target_2790,v30,z15,My_Mechanism_1\WObj:=Workobject_1;
        WaitTime 0.5;
        MoveL Target_2800,v30,z15,My_Mechanism_1\WObj:=Workobject_1;
        MoveL Target_2810,v30,z15,My_Mechanism_1\WObj:=Workobject_1;
        MoveL Target_2820,v30,z15,My_Mechanism_1\WObj:=Workobject_1;
        MoveL Target_2830,v30,z15,My_Mechanism_1\WObj:=Workobject_1;
        MoveL Target_2840,v30,z15,My_Mechanism_1\WObj:=Workobject_1;
        MoveL Target_2850,v30,z15,My_Mechanism_1\WObj:=Workobject_1;
        MoveL Target_2860,v30,z15,My_Mechanism_1\WObj:=Workobject_1;
        MoveL Target_2870,v30,z15,My_Mechanism_1\WObj:=Workobject_1;
        MoveL Target_2880,v30,z15,My_Mechanism_1\WObj:=Workobject_1;
        MoveL Target_2890,v30,z15,My_Mechanism_1\WObj:=Workobject_1;
        MoveL Target_2900,v30,z15,My_Mechanism_1\WObj:=Workobject_1;
        MoveL Target_2910,v30,z15,My_Mechanism_1\WObj:=Workobject_1;
        MoveL Target_2920,v30,z15,My_Mechanism_1\WObj:=Workobject_1;
        MoveL Target_2930,v30,z15,My_Mechanism_1\WObj:=Workobject_1;
        MoveL Target_2940,v30,z15,My_Mechanism_1\WObj:=Workobject_1;
        MoveL Target_2950,v30,z15,My_Mechanism_1\WObj:=Workobject_1;
        MoveL Target_2960,v30,z15,My_Mechanism_1\WObj:=Workobject_1;
        MoveL Target_2970,v30,z15,My_Mechanism_1\WObj:=Workobject_1;
        MoveL Target_2980,v30,z15,My_Mechanism_1\WObj:=Workobject_1;
        MoveL Target_2990,v30,z15,My_Mechanism_1\WObj:=Workobject_1;
        MoveL Target_3000,v30,z15,My_Mechanism_1\WObj:=Workobject_1;
        MoveL Target_3010,v30,z15,My_Mechanism_1\WObj:=Workobject_1;
        MoveL Target_3020,v30,z15,My_Mechanism_1\WObj:=Workobject_1;
        MoveL Target_3030,v30,z15,My_Mechanism_1\WObj:=Workobject_1;
        MoveL Target_3040,v30,z15,My_Mechanism_1\WObj:=Workobject_1;
        MoveL Target_3050,v30,z15,My_Mechanism_1\WObj:=Workobject_1;
        MoveL Target_3060,v30,z15,My_Mechanism_1\WObj:=Workobject_1;
        MoveL Target_3070,v30,z15,My_Mechanism_1\WObj:=Workobject_1;
        MoveL Target_3080,v30,z15,My_Mechanism_1\WObj:=Workobject_1;
        MoveL Target_3090,v30,z15,My_Mechanism_1\WObj:=Workobject_1;
        MoveL Target_3100,v30,z15,My_Mechanism_1\WObj:=Workobject_1;
        MoveL Target_3110,v30,z15,My_Mechanism_1\WObj:=Workobject_1;
        MoveL Target_3120,v30,z15,My_Mechanism_1\WObj:=Workobject_1;
        MoveL Target_3130,v30,z15,My_Mechanism_1\WObj:=Workobject_1;
        MoveL Target_3140,v30,z15,My_Mechanism_1\WObj:=Workobject_1;
        MoveL Target_3150,v30,z15,My_Mechanism_1\WObj:=Workobject_1;
        MoveL Target_3160,v30,z15,My_Mechanism_1\WObj:=Workobject_1;
        MoveL Target_3170,v30,z15,My_Mechanism_1\WObj:=Workobject_1;
        MoveL Target_3180,v30,z15,My_Mechanism_1\WObj:=Workobject_1;
        WaitTime 0.5;
    ENDPROC
    PROC Stinks_t()
        MoveL Target_3190,v30,z15,My_Mechanism_1\WObj:=Workobject_1;
        WaitTime 0.5;
        MoveL Target_3200,v30,z15,My_Mechanism_1\WObj:=Workobject_1;
        MoveL Target_3210,v30,z15,My_Mechanism_1\WObj:=Workobject_1;
        MoveL Target_3220,v30,z15,My_Mechanism_1\WObj:=Workobject_1;
        MoveL Target_3230,v30,z15,My_Mechanism_1\WObj:=Workobject_1;
        MoveL Target_3240,v30,z15,My_Mechanism_1\WObj:=Workobject_1;
        MoveL Target_3250,v30,z15,My_Mechanism_1\WObj:=Workobject_1;
        MoveL Target_3260,v30,z15,My_Mechanism_1\WObj:=Workobject_1;
        MoveL Target_3270,v30,z15,My_Mechanism_1\WObj:=Workobject_1;
        MoveL Target_3280,v30,z15,My_Mechanism_1\WObj:=Workobject_1;
        MoveL Target_3290,v30,z15,My_Mechanism_1\WObj:=Workobject_1;
        MoveL Target_3300,v30,z15,My_Mechanism_1\WObj:=Workobject_1;
        MoveL Target_3310,v30,z15,My_Mechanism_1\WObj:=Workobject_1;
        MoveL Target_3320,v30,z15,My_Mechanism_1\WObj:=Workobject_1;
        MoveL Target_3330,v30,z15,My_Mechanism_1\WObj:=Workobject_1;
        MoveL Target_3340,v30,z15,My_Mechanism_1\WObj:=Workobject_1;
        MoveL Target_3350,v30,z15,My_Mechanism_1\WObj:=Workobject_1;
        MoveL Target_3360,v30,z15,My_Mechanism_1\WObj:=Workobject_1;
        MoveL Target_3370,v30,z15,My_Mechanism_1\WObj:=Workobject_1;
        MoveL Target_3380,v30,z15,My_Mechanism_1\WObj:=Workobject_1;
        MoveL Target_3390,v30,z15,My_Mechanism_1\WObj:=Workobject_1;
        MoveL Target_3400,v30,z15,My_Mechanism_1\WObj:=Workobject_1;
        WaitTime 0.5;
    ENDPROC
    PROC Stinks_i()
        MoveL Target_3410,v30,z15,My_Mechanism_1\WObj:=Workobject_1;
        WaitTime 0.5;
        MoveL Target_3420,v30,z15,My_Mechanism_1\WObj:=Workobject_1;
        MoveL Target_3430,v30,z15,My_Mechanism_1\WObj:=Workobject_1;
        MoveL Target_3440,v30,z15,My_Mechanism_1\WObj:=Workobject_1;
        MoveL Target_3450,v30,z15,My_Mechanism_1\WObj:=Workobject_1;
        MoveL Target_3460,v30,z15,My_Mechanism_1\WObj:=Workobject_1;
        MoveL Target_3470,v30,z15,My_Mechanism_1\WObj:=Workobject_1;
        MoveL Target_3480,v30,z15,My_Mechanism_1\WObj:=Workobject_1;
        MoveL Target_3490,v30,z15,My_Mechanism_1\WObj:=Workobject_1;
        MoveL Target_3500,v30,z15,My_Mechanism_1\WObj:=Workobject_1;
        WaitTime 0.5;
        MoveL LiftPoint_stinks,v30,z15,My_Mechanism_1\WObj:=Workobject_1;
        Stink_i_dot;
    ENDPROC
    PROC Stink_i_dot()
        MoveL Target_3510,v30,z15,My_Mechanism_1\WObj:=Workobject_1;
        WaitTime 0.5;
        MoveL Target_3520,v30,z15,My_Mechanism_1\WObj:=Workobject_1;
        MoveL Target_3530,v30,z15,My_Mechanism_1\WObj:=Workobject_1;
        MoveL Target_3540,v30,z15,My_Mechanism_1\WObj:=Workobject_1;
        MoveL Target_3550,v30,z15,My_Mechanism_1\WObj:=Workobject_1;
        MoveL Target_3560,v30,z15,My_Mechanism_1\WObj:=Workobject_1;
        MoveL Target_3570,v30,z15,My_Mechanism_1\WObj:=Workobject_1;
        MoveL Target_3580,v30,z15,My_Mechanism_1\WObj:=Workobject_1;
        MoveL Target_3590,v30,z15,My_Mechanism_1\WObj:=Workobject_1;
        WaitTime 0.5;
    ENDPROC
    PROC Stinks_n()
        MoveL Target_3600,v30,z15,My_Mechanism_1\WObj:=Workobject_1;
        WaitTime 0.5;
        MoveL Target_3610,v30,z15,My_Mechanism_1\WObj:=Workobject_1;
        MoveL Target_3620,v30,z15,My_Mechanism_1\WObj:=Workobject_1;
        MoveL Target_3630,v30,z15,My_Mechanism_1\WObj:=Workobject_1;
        MoveL Target_3640,v30,z15,My_Mechanism_1\WObj:=Workobject_1;
        MoveL Target_3650,v30,z15,My_Mechanism_1\WObj:=Workobject_1;
        MoveL Target_3660,v30,z15,My_Mechanism_1\WObj:=Workobject_1;
        MoveL Target_3670,v30,z15,My_Mechanism_1\WObj:=Workobject_1;
        MoveL Target_3680,v30,z15,My_Mechanism_1\WObj:=Workobject_1;
        MoveL Target_3690,v30,z15,My_Mechanism_1\WObj:=Workobject_1;
        MoveL Target_3700,v30,z15,My_Mechanism_1\WObj:=Workobject_1;
        MoveL Target_3710,v30,z15,My_Mechanism_1\WObj:=Workobject_1;
        MoveL Target_3720,v30,z15,My_Mechanism_1\WObj:=Workobject_1;
        MoveL Target_3730,v30,z15,My_Mechanism_1\WObj:=Workobject_1;
        MoveL Target_3740,v30,z15,My_Mechanism_1\WObj:=Workobject_1;
        MoveL Target_3750,v30,z15,My_Mechanism_1\WObj:=Workobject_1;
        MoveL Target_3760,v30,z15,My_Mechanism_1\WObj:=Workobject_1;
        MoveL Target_3770,v30,z15,My_Mechanism_1\WObj:=Workobject_1;
        MoveL Target_3780,v30,z15,My_Mechanism_1\WObj:=Workobject_1;
        MoveL Target_3790,v30,z15,My_Mechanism_1\WObj:=Workobject_1;
        MoveL Target_3800,v30,z15,My_Mechanism_1\WObj:=Workobject_1;
        MoveL Target_3810,v30,z15,My_Mechanism_1\WObj:=Workobject_1;
        MoveL Target_3820,v30,z15,My_Mechanism_1\WObj:=Workobject_1;
        MoveL Target_3830,v30,z15,My_Mechanism_1\WObj:=Workobject_1;
        WaitTime 0.5;
    ENDPROC
    PROC Stinks_k()
        MoveL Target_3840,v30,z15,My_Mechanism_1\WObj:=Workobject_1;
        WaitTime 0.5;
        MoveL Target_3850,v30,z15,My_Mechanism_1\WObj:=Workobject_1;
        MoveL Target_3860,v30,z15,My_Mechanism_1\WObj:=Workobject_1;
        MoveL Target_3870,v30,z15,My_Mechanism_1\WObj:=Workobject_1;
        MoveL Target_3880,v30,z15,My_Mechanism_1\WObj:=Workobject_1;
        MoveL Target_3890,v30,z15,My_Mechanism_1\WObj:=Workobject_1;
        MoveL Target_3900,v30,z15,My_Mechanism_1\WObj:=Workobject_1;
        MoveL Target_3910,v30,z15,My_Mechanism_1\WObj:=Workobject_1;
        MoveL Target_3920,v30,z15,My_Mechanism_1\WObj:=Workobject_1;
        MoveL Target_3930,v30,z15,My_Mechanism_1\WObj:=Workobject_1;
        MoveL Target_3940,v30,z15,My_Mechanism_1\WObj:=Workobject_1;
        MoveL Target_3950,v30,z15,My_Mechanism_1\WObj:=Workobject_1;
        MoveL Target_3960,v30,z15,My_Mechanism_1\WObj:=Workobject_1;
        MoveL Target_3970,v30,z15,My_Mechanism_1\WObj:=Workobject_1;
        MoveL Target_3980,v30,z15,My_Mechanism_1\WObj:=Workobject_1;
        MoveL Target_3990,v30,z15,My_Mechanism_1\WObj:=Workobject_1;
        MoveL Target_4000,v30,z15,My_Mechanism_1\WObj:=Workobject_1;
        MoveL Target_4010,v30,z15,My_Mechanism_1\WObj:=Workobject_1;
        MoveL Target_4020,v30,z15,My_Mechanism_1\WObj:=Workobject_1;
        MoveL Target_4030,v30,z15,My_Mechanism_1\WObj:=Workobject_1;
        MoveL Target_4040,v30,z15,My_Mechanism_1\WObj:=Workobject_1;
        MoveL Target_4050,v30,z15,My_Mechanism_1\WObj:=Workobject_1;
        WaitTime 0.5;
    ENDPROC
    PROC Stinks_s_2()
        MoveL Target_4060,v30,z15,My_Mechanism_1\WObj:=Workobject_1;
        WaitTime 0.5;
        MoveL Target_4070,v30,z15,My_Mechanism_1\WObj:=Workobject_1;
        MoveL Target_4080,v30,z15,My_Mechanism_1\WObj:=Workobject_1;
        MoveL Target_4090,v30,z15,My_Mechanism_1\WObj:=Workobject_1;
        MoveL Target_4100,v30,z15,My_Mechanism_1\WObj:=Workobject_1;
        MoveL Target_4110,v30,z15,My_Mechanism_1\WObj:=Workobject_1;
        MoveL Target_4120,v30,z15,My_Mechanism_1\WObj:=Workobject_1;
        MoveL Target_4130,v30,z15,My_Mechanism_1\WObj:=Workobject_1;
        MoveL Target_4140,v30,z15,My_Mechanism_1\WObj:=Workobject_1;
        MoveL Target_4150,v30,z15,My_Mechanism_1\WObj:=Workobject_1;
        MoveL Target_4160,v30,z15,My_Mechanism_1\WObj:=Workobject_1;
        MoveL Target_4170,v30,z15,My_Mechanism_1\WObj:=Workobject_1;
        MoveL Target_4180,v30,z15,My_Mechanism_1\WObj:=Workobject_1;
        MoveL Target_4190,v30,z15,My_Mechanism_1\WObj:=Workobject_1;
        MoveL Target_4200,v30,z15,My_Mechanism_1\WObj:=Workobject_1;
        MoveL Target_4210,v30,z15,My_Mechanism_1\WObj:=Workobject_1;
        MoveL Target_4220,v30,z15,My_Mechanism_1\WObj:=Workobject_1;
        MoveL Target_4230,v30,z15,My_Mechanism_1\WObj:=Workobject_1;
        MoveL Target_4240,v30,z15,My_Mechanism_1\WObj:=Workobject_1;
        MoveL Target_4250,v30,z15,My_Mechanism_1\WObj:=Workobject_1;
        MoveL Target_4260,v30,z15,My_Mechanism_1\WObj:=Workobject_1;
        MoveL Target_4270,v30,z15,My_Mechanism_1\WObj:=Workobject_1;
        MoveL Target_4280,v30,z15,My_Mechanism_1\WObj:=Workobject_1;
        MoveL Target_4290,v30,z15,My_Mechanism_1\WObj:=Workobject_1;
        MoveL Target_4300,v30,z15,My_Mechanism_1\WObj:=Workobject_1;
        MoveL Target_4310,v30,z15,My_Mechanism_1\WObj:=Workobject_1;
        MoveL Target_4320,v30,z15,My_Mechanism_1\WObj:=Workobject_1;
        MoveL Target_4330,v30,z15,My_Mechanism_1\WObj:=Workobject_1;
        MoveL Target_4340,v30,z15,My_Mechanism_1\WObj:=Workobject_1;
        MoveL Target_4350,v30,z15,My_Mechanism_1\WObj:=Workobject_1;
        MoveL Target_4360,v30,z15,My_Mechanism_1\WObj:=Workobject_1;
        WaitTime 0.5;
    ENDPROC
ENDMODULE

